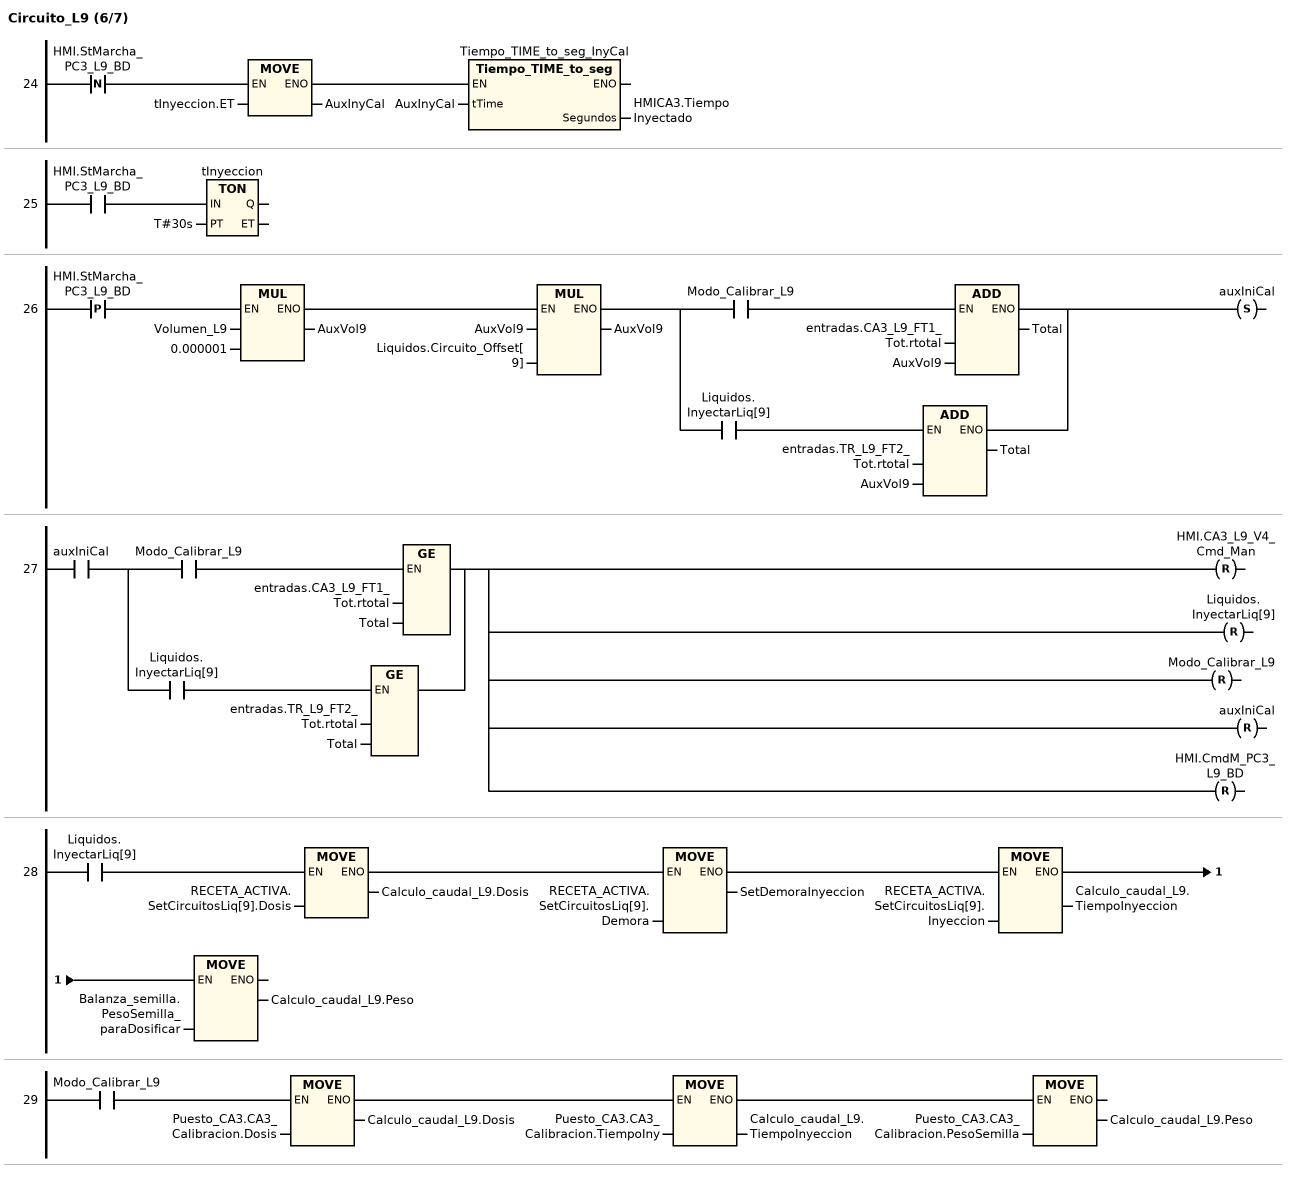
// NETWORK 24
_ft1(CLK := HMI.StMarcha_PC3_L9_BD);
_w8 := _ft1.Q;
IF _w8 THEN AuxInyCal := tInyeccion.ET; END_IF
IF _w8 THEN
    Tiempo_TIME_to_seg_InyCal(tTime := AuxInyCal, Segundos => HMICA3.TiempoInyectado); // Tiempo_TIME_to_seg
END_IF

// NETWORK 25
tInyeccion(IN := HMI.StMarcha_PC3_L9_BD, PT := T#30s); // TON

// NETWORK 26
_rt1(CLK := HMI.StMarcha_PC3_L9_BD);
_w9 := _rt1.Q;
IF _w9 THEN AuxVol9 := Volumen_L9 * 0.000001; END_IF
IF _w9 THEN AuxVol9 := AuxVol9 * Liquidos.Circuito_Offset[9]; END_IF
IF _w9 AND Modo_Calibrar_L9 THEN Total := entradas.CA3_L9_FT1_Tot.rtotal + AuxVol9; END_IF
IF _w9 AND Liquidos.InyectarLiq[9] THEN Total := entradas.TR_L9_FT2_Tot.rtotal + AuxVol9; END_IF
auxIniCal S= _w9 AND Modo_Calibrar_L9 OR _w9 AND Liquidos.InyectarLiq[9];

// NETWORK 27
_w10 := auxIniCal AND Modo_Calibrar_L9 AND entradas.CA3_L9_FT1_Tot.rtotal >= Total OR auxIniCal AND Liquidos.InyectarLiq[9] AND entradas.TR_L9_FT2_Tot.rtotal >= Total;
HMI.CA3_L9_V4_Cmd_Man R= _w10;
Liquidos.InyectarLiq[9] R= _w10;
Modo_Calibrar_L9 R= _w10;
auxIniCal R= _w10;
HMI.CmdM_PC3_L9_BD R= _w10;

// NETWORK 28
_w11 := Liquidos.InyectarLiq[9];
IF _w11 THEN Calculo_caudal_L9.Dosis := RECETA_ACTIVA.SetCircuitosLiq[9].Dosis; END_IF
IF _w11 THEN SetDemoraInyeccion := RECETA_ACTIVA.SetCircuitosLiq[9].Demora; END_IF
IF _w11 THEN Calculo_caudal_L9.TiempoInyeccion := RECETA_ACTIVA.SetCircuitosLiq[9].Inyeccion; END_IF
IF _w11 THEN Calculo_caudal_L9.Peso := Balanza_semilla.PesoSemilla_paraDosificar; END_IF

// NETWORK 29
_w12 := Modo_Calibrar_L9;
IF _w12 THEN Calculo_caudal_L9.Dosis := Puesto_CA3.CA3_Calibracion.Dosis; END_IF
IF _w12 THEN Calculo_caudal_L9.TiempoInyeccion := Puesto_CA3.CA3_Calibracion.TiempoIny; END_IF
IF _w12 THEN Calculo_caudal_L9.Peso := Puesto_CA3.CA3_Calibracion.PesoSemilla; END_IF

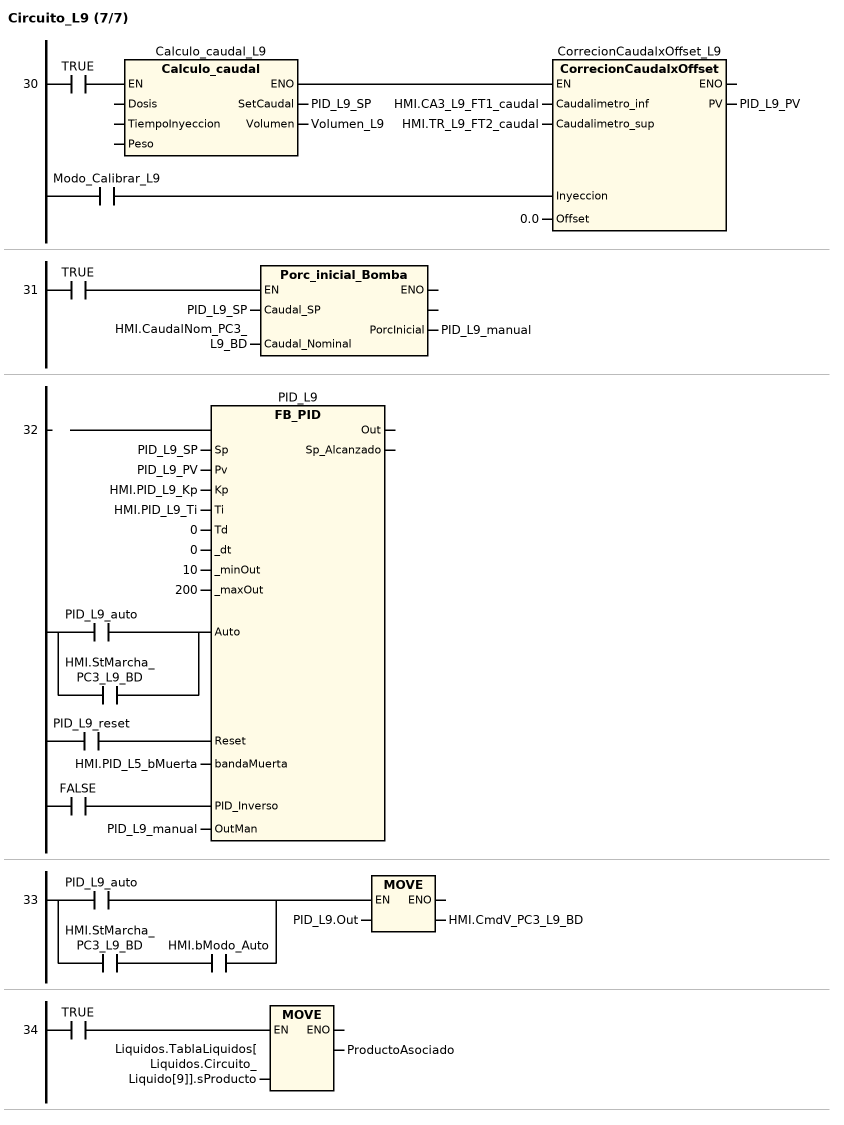
// NETWORK 30
Calculo_caudal_L9(SetCaudal => PID_L9_SP, Volumen => Volumen_L9); // Calculo_caudal
CorrecionCaudalxOffset_L9(
    Caudalimetro_inf := HMI.CA3_L9_FT1_caudal,
    Caudalimetro_sup := HMI.TR_L9_FT2_caudal,
    Inyeccion := Modo_Calibrar_L9,
    Offset := 0.0,
    PV => PID_L9_PV); // CorrecionCaudalxOffset

// NETWORK 31
Porc_inicial_Bomba(Caudal_SP := PID_L9_SP, Caudal_Nominal := HMI.CaudalNom_PC3_L9_BD, PorcInicial => PID_L9_manual);

// NETWORK 32
PID_L9(
    Sp := PID_L9_SP,
    Pv := PID_L9_PV,
    Kp := HMI.PID_L9_Kp,
    Ti := HMI.PID_L9_Ti,
    Td := 0,
    _dt := 0,
    _minOut := 10,
    _maxOut := 200,
    Auto := PID_L9_auto OR HMI.StMarcha_PC3_L9_BD,
    Reset := PID_L9_reset,
    bandaMuerta := HMI.PID_L5_bMuerta,
    PID_Inverso := FALSE,
    OutMan := PID_L9_manual); // FB_PID

// NETWORK 33
IF PID_L9_auto OR HMI.StMarcha_PC3_L9_BD AND HMI.bModo_Auto THEN HMI.CmdV_PC3_L9_BD := PID_L9.Out; END_IF

// NETWORK 34
ProductoAsociado := Liquidos.TablaLiquidos[Liquidos.Circuito_Liquido[9]].sProducto;

END_PROGRAM

// ---- POUs/Puesto_Calibracion_3/Puesto_CA3.TcPOU
PROGRAM Puesto_CA3
VAR
	Balanza_CA3: Balanza;
	dHS:DINT;
	Cmd_Full: R_TRIG;
	TmrLabelFinalizado: TON;
	AuxFinCalibrar:BOOL;
	CA3_Calibracion: Calibracion_Liq_calc;
	Tarar_balanza :BOOL;
	Offset_ref3:REAL;
	Inyectar_ref3:BOOL;
	InicioCal_ref3:BOOL;
	Offset_ref: REAL;
	Inyectar_ref: BOOL;
	InicioCal_ref: BOOL;

	UltimaCalibracao: UDINT;
	VazaoMax: REAL;
	VazaoMaxExcedida: BOOL;
END_VAR

//Indica a ultima calibração da linha selecionada
UltimaCalibracao := HMI.UltimasCalibracoes[HMI.iCircuito_a_calibrar];


Balanza_CA3(
	wStatus:=Entradas.CA3_WT1_wStatus , 
	rValue_REAL:=Entradas.CA3_WT1_rValue_REAL , 
	nValue_DINT:=Entradas.CA3_WT1_nValue_DINT , 
	nValue_Supply:=dHS , 
	nValue_Bridge:=dHS , 
	stEcSlaveAmsNetAdr:=Entradas.CA3_WT1_stEcSlaveAmsNetAdr , 
	bWcState:=Entradas.CA3_WT1_bWcState , 
	wState:=Entradas.CA3_WT1_wState , 
	bCmd_FullCalibration:=HMI.bCmd_Full_WT_CA3 , 
	bCmd_ZeroCalibration:=HMI.bCmd_Zero_WT_CA3 , 
	bCmd_Tara:=Tarar_balanza , 
	bCmd_LoadReference:=HMI.bCmd_LoadReference_WT_CA3 ,
	fLoadReference:=(HMI.rPesoPatron_WT_CA3)/1000,
	wControl=>Salidas.CA3_WT1_wControl );

	TmrLabelFinalizado(IN:= HMI.bCmd_Full_WT_CA3 , PT:=T#10S , Q=> , ET=> );	
	
	HMI.bCmd_LoadReference_WT_CA3:=FALSE;
	HMI.bCmd_Zero_WT_CA3:=FALSE;
	HMI.bCmd_Full_WT_CA3:=FALSE;
	Tarar_balanza:=FALSE;
	Cmd_Full(CLK:=TmrLabelFinalizado.Q , Q=> );
	IF 	Cmd_Full.Q THEN
		HMI.bCalibrado_WT_CA3:=TRUE;
	END_IF	
/////////////////
IF (8<HMI.iCircuito_a_calibrar AND HMI.iCircuito_a_calibrar<13) THEN
//
/////////
CASE HMI.iCircuito_a_calibrar OF
	9:	Offset_ref:=Liquidos.Circuito_Offset[9];
		Inyectar_ref:=circuito_L9.Modo_Calibrar_L9;
		InicioCal_ref:=HMICA3.Inicio_calibracion;
		HMICA3.VolumenPedido_calibracion:=circuito_L9.Volumen_L9;
	10:	Offset_ref:=Liquidos.Circuito_Offset[10];
		Inyectar_ref:=circuito_L10.Modo_Calibrar_L10;
		InicioCal_ref:=HMICA3.Inicio_calibracion;
		HMICA3.VolumenPedido_calibracion:=circuito_L10.Volumen_L10;	
	11:	Offset_ref:=Liquidos.Circuito_Offset[11];
		Inyectar_ref:=circuito_L11.Modo_Calibrar_L11;
		InicioCal_ref:=HMICA3.Inicio_calibracion;
		HMICA3.VolumenPedido_calibracion:=circuito_L11.Volumen_L11;
	12:	Offset_ref:=Liquidos.Circuito_Offset[12];
		Inyectar_ref:=circuito_L12.Modo_Calibrar_L12;
		InicioCal_ref:=HMICA3.Inicio_calibracion;
		HMICA3.VolumenPedido_calibracion:=circuito_L12.Volumen_L12;	
		
		ELSE
	;		
END_CASE
CA3_Calibracion(
	Dosis:=HMICA3.Dosis_calibracion , 
	PesoSemilla:=HMICA3.Peso_calibracion,
	Tolerancia:=HMICA3.Tolerancia_calibracion , 
	PesoBalanza:=Entradas.CA3_WT1_rValue_REAL ,
	mlPedido:= HMICA3.VolumenPedido_calibracion,
	PesoEspec:=Puesto_CA1.PesoEspec , 
	Offset:=Offset_ref ,
	TiempoIny:=HMICA3.TInyeccion_calibracion , 
	Vol_Probeta:=(HMICA3.VolMaxProbeta_calibracion*1000) , 
	Pausa:=HMICA3.Pausa_calibracion , 
	Dosificar=> , 
	Probeta_Llena:=HMICA3.VaciarProbeta_calibracion , 
	Inyectar:=Inyectar_ref, 
	ml:=HMICA3.Volumen_calibracion, 
	Tiempo:=HMICA3.Tiempo_calibracion , 
	InicioCal:= InicioCal_ref, 
	Continuar:=HMICA3.Continuar_calibracion , 
	Tarar:=Tarar_balanza,
	Finalizado:=HMICA3.Fin_calibracion,
	mlProbeta=>HMICA3.Vol_enProbeta , 
	TiempoInyectado:=HMICA3.TiempoInyectado,
	Error_promedio=> HMICA3.Error_promedio, );
//
CASE HMI.iCircuito_a_calibrar OF
	9:	Liquidos.Circuito_Offset[9]:=Offset_ref;//Offset_ref
		circuito_L9.Modo_Calibrar_L9:=Inyectar_ref;//Inyectar_ref
		HMICA3.Inicio_calibracion:=InicioCal_ref;
		VazaoMax := HMI.CaudalNom_PC3_L9_BD;
	10:	Liquidos.Circuito_Offset[10]:=Offset_ref;//Offset_ref
		circuito_L10.Modo_Calibrar_L10:=Inyectar_ref;//Inyectar_ref
		HMICA3.Inicio_calibracion:=InicioCal_ref;
		VazaoMax := HMI.CaudalNom_PC3_L10_BD;
	11:	Liquidos.Circuito_Offset[11]:=Offset_ref;//Offset_ref
		circuito_L11.Modo_Calibrar_L11:=Inyectar_ref;//Inyectar_ref
		HMICA3.Inicio_calibracion:=InicioCal_ref;
		VazaoMax := HMI.CaudalNom_PC3_L11_BD;
	12:	Liquidos.Circuito_Offset[12]:=Offset_ref;//Offset_ref
		circuito_L12.Modo_Calibrar_L12:=Inyectar_ref;//Inyectar_ref
		HMICA3.Inicio_calibracion:=InicioCal_ref;
		VazaoMax := HMI.CaudalNom_PC3_L12_BD;
		
		ELSE
	;		
END_CASE	
END_IF	

IF HMICA3.TInyeccion_calibracion > 0 THEN
	IF (HMICA3.Dosis_calibracion*HMICA3.Peso_calibracion/100)/TO_REAL(HMICA3.TInyeccion_calibracion) > VazaoMax THEN
		VazaoMaxExcedida := TRUE;
	ELSE
		VazaoMaxExcedida := FALSE;
	END_IF
END_IF

END_PROGRAM

// ---- POUs/Puesto_Calibracion_3/Circuito_L10.TcPOU
PROGRAM Circuito_L10
VAR_INPUT
	Modo_Calibrar_L10: BOOL;
END_VAR
VAR
		fbBomba_L10 :Equipo_Motor_ATV320;
		ControlValv_ioLink_V1:ControlValv_ioLink;
		ControlValv_ioLink_V2: ControlValv_ioLink;
		ControlValv_ioLink_V3: ControlValv_ioLink;
		ControlValv_ioLink_V4: ControlValv_ioLink;
		Falla_L10_V1:BOOL;
		Falla_L10_V2:BOOL;
		Falla_L10_V3:BOOL;
		Falla_L10_V4:BOOL;
	Balanza_PU3_WT10: Balanza;
		dHS:DINT;
		TOF_calibradoIBC: TOF;
		PID_L10_SP:REAL;
		PID_L10_auto:BOOL;
		PID_L10_reset:BOOL;
		PID_L10_manual:REAL;
		PID_L10_bMuerta:REAL := 5;
		PID_L10_Kp:REAL := 0.1;
		PID_L10_Ti:REAL := 100;
		PID_L10_PV:REAL;
		Dosis_L10	:REAL;
		TiempoInyeccion_L10	:DINT;
		Peso	:REAL;
		Offset_L10:REAL;
		Inyeccion_L10:BOOL;

		Volumen_L10:REAL;
		Calculo_caudal_L10: Calculo_caudal;
		CorrecionCaudalxOffset_L10: CorrecionCaudalxOffset;
		tInyeccion: TON;
		Total :REAL;
		Totalant	:REAL;
		auxIniCal:BOOL;
		AuxVol10:REAL;
		TDemoraInyectar: TON;
		SetDemoraInyeccion: REAL;
		Tiempo_seg_to_TIME_DemoraInyec: Tiempo_seg_to_TIME;
		AuxTDemoraInyec: TIME;
		PID_L10: FB_PID;
		Tiempo_TIME_to_seg_InyCal: Tiempo_TIME_to_seg;
		AuxInyCal:TIME;
	ProductoAsociado: STRING;
	Lavagem_Circuito10: Lavagem;
END_VAR
VAR PERSISTENT
	UltimaCalibracao	:UDINT;	//Data e hora da ultima calibração
END_VAR
VAR // added by the converter: edge detectors and wires of the graphical bodies
    _w1, _w2, _w3, _w4, _w5, _w6, _w7, _w8, _w9, _w10, _w11, _w12 : BOOL;
    _ft1 : F_TRIG;
    _rt1 : R_TRIG;
END_VAR

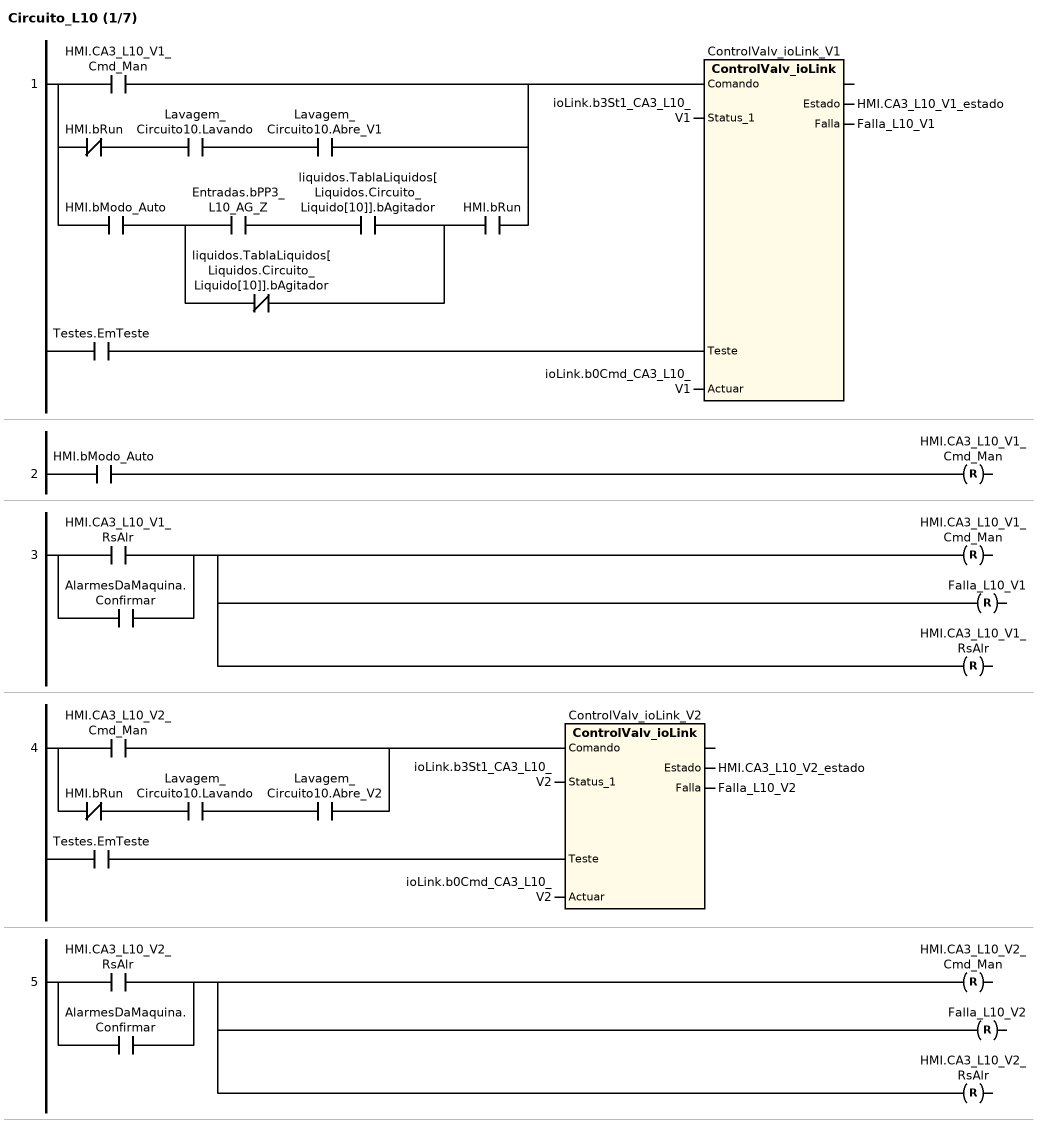
// NETWORK 1
ControlValv_ioLink_V1(
    Comando := HMI.CA3_L10_V1_Cmd_Man OR NOT HMI.bRun AND Lavagem_Circuito10.Lavando AND Lavagem_Circuito10.Abre_V1 OR HMI.bModo_Auto AND (Entradas.bPP3_L10_AG_Z AND (liquidos.TablaLiquidos[Liquidos.Circuito_Liquido[10]].bAgitador) OR NOT (liquidos.TablaLiquidos[Liquidos.Circuito_Liquido[10]].bAgitador)) AND HMI.bRun,
    Status_1 := ioLink.b3St1_CA3_L10_V1,
    Teste := Testes.EmTeste,
    Actuar := ioLink.b0Cmd_CA3_L10_V1,
    Estado => HMI.CA3_L10_V1_estado,
    Falla => Falla_L10_V1); // ControlValv_ioLink

// NETWORK 2
HMI.CA3_L10_V1_Cmd_Man R= HMI.bModo_Auto;

// NETWORK 3
_w1 := HMI.CA3_L10_V1_RsAlr OR AlarmesDaMaquina.Confirmar;
HMI.CA3_L10_V1_Cmd_Man R= _w1;
Falla_L10_V1 R= _w1;
HMI.CA3_L10_V1_RsAlr R= _w1;

// NETWORK 4
ControlValv_ioLink_V2(
    Comando := HMI.CA3_L10_V2_Cmd_Man OR NOT HMI.bRun AND Lavagem_Circuito10.Lavando AND Lavagem_Circuito10.Abre_V2,
    Status_1 := ioLink.b3St1_CA3_L10_V2,
    Teste := Testes.EmTeste,
    Actuar := ioLink.b0Cmd_CA3_L10_V2,
    Estado => HMI.CA3_L10_V2_estado,
    Falla => Falla_L10_V2); // ControlValv_ioLink

// NETWORK 5
_w2 := HMI.CA3_L10_V2_RsAlr OR AlarmesDaMaquina.Confirmar;
HMI.CA3_L10_V2_Cmd_Man R= _w2;
Falla_L10_V2 R= _w2;
HMI.CA3_L10_V2_RsAlr R= _w2;

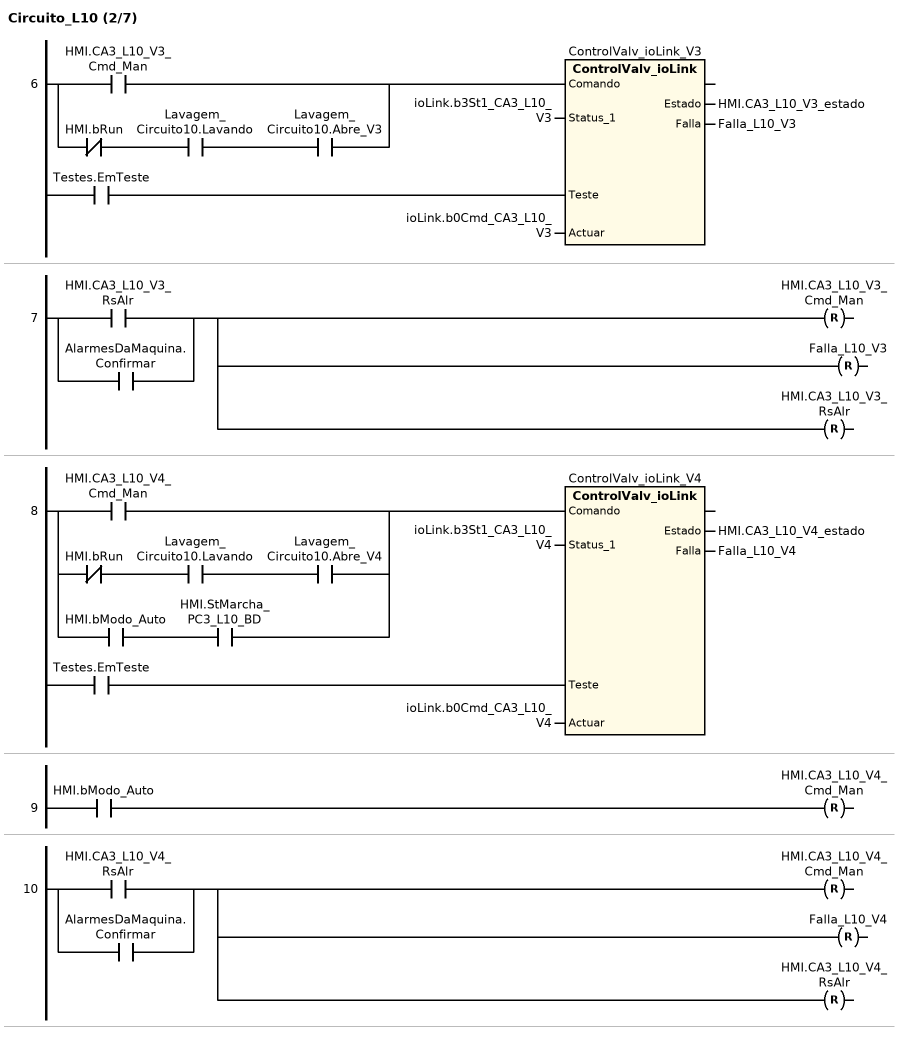
// NETWORK 6
ControlValv_ioLink_V3(
    Comando := HMI.CA3_L10_V3_Cmd_Man OR NOT HMI.bRun AND Lavagem_Circuito10.Lavando AND Lavagem_Circuito10.Abre_V3,
    Status_1 := ioLink.b3St1_CA3_L10_V3,
    Teste := Testes.EmTeste,
    Actuar := ioLink.b0Cmd_CA3_L10_V3,
    Estado => HMI.CA3_L10_V3_estado,
    Falla => Falla_L10_V3); // ControlValv_ioLink

// NETWORK 7
_w3 := HMI.CA3_L10_V3_RsAlr OR AlarmesDaMaquina.Confirmar;
HMI.CA3_L10_V3_Cmd_Man R= _w3;
Falla_L10_V3 R= _w3;
HMI.CA3_L10_V3_RsAlr R= _w3;

// NETWORK 8
ControlValv_ioLink_V4(
    Comando := HMI.CA3_L10_V4_Cmd_Man OR NOT HMI.bRun AND Lavagem_Circuito10.Lavando AND Lavagem_Circuito10.Abre_V4 OR HMI.bModo_Auto AND HMI.StMarcha_PC3_L10_BD,
    Status_1 := ioLink.b3St1_CA3_L10_V4,
    Teste := Testes.EmTeste,
    Actuar := ioLink.b0Cmd_CA3_L10_V4,
    Estado => HMI.CA3_L10_V4_estado,
    Falla => Falla_L10_V4); // ControlValv_ioLink

// NETWORK 9
HMI.CA3_L10_V4_Cmd_Man R= HMI.bModo_Auto;

// NETWORK 10
_w4 := HMI.CA3_L10_V4_RsAlr OR AlarmesDaMaquina.Confirmar;
HMI.CA3_L10_V4_Cmd_Man R= _w4;
Falla_L10_V4 R= _w4;
HMI.CA3_L10_V4_RsAlr R= _w4;

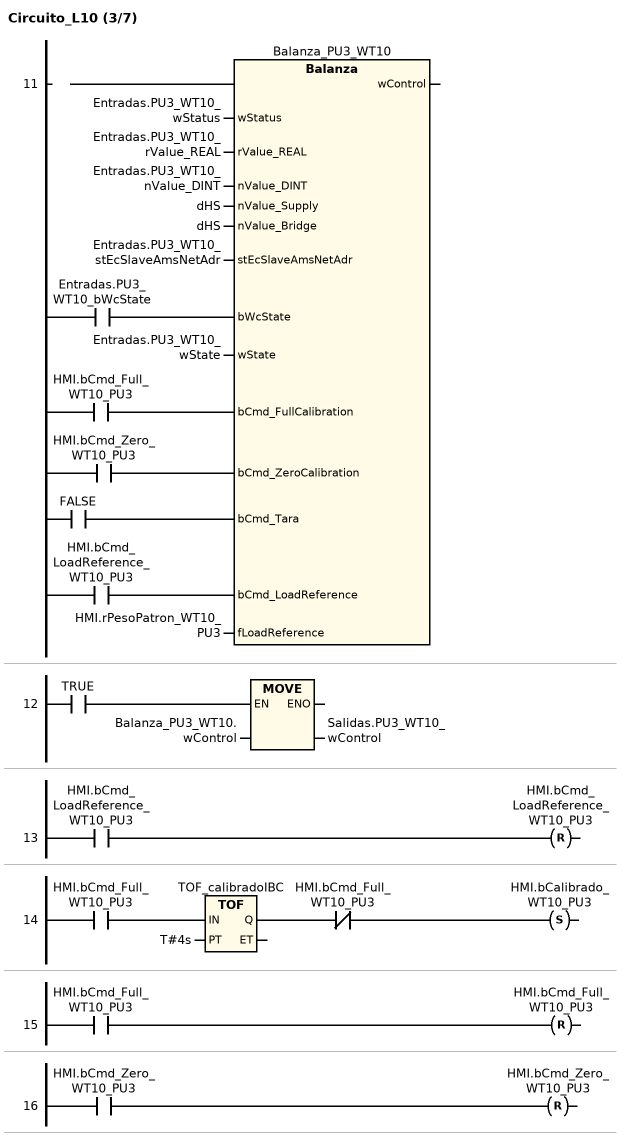
// NETWORK 11
Balanza_PU3_WT10(
    wStatus := Entradas.PU3_WT10_wStatus,
    rValue_REAL := Entradas.PU3_WT10_rValue_REAL,
    nValue_DINT := Entradas.PU3_WT10_nValue_DINT,
    nValue_Supply := dHS,
    nValue_Bridge := dHS,
    stEcSlaveAmsNetAdr := Entradas.PU3_WT10_stEcSlaveAmsNetAdr,
    bWcState := Entradas.PU3_WT10_bWcState,
    wState := Entradas.PU3_WT10_wState,
    bCmd_FullCalibration := HMI.bCmd_Full_WT10_PU3,
    bCmd_ZeroCalibration := HMI.bCmd_Zero_WT10_PU3,
    bCmd_Tara := FALSE,
    bCmd_LoadReference := HMI.bCmd_LoadReference_WT10_PU3,
    fLoadReference := HMI.rPesoPatron_WT10_PU3); // Balanza

// NETWORK 12
Salidas.PU3_WT10_wControl := Balanza_PU3_WT10.wControl;

// NETWORK 13
HMI.bCmd_LoadReference_WT10_PU3 R= HMI.bCmd_LoadReference_WT10_PU3;

// NETWORK 14
TOF_calibradoIBC(IN := HMI.bCmd_Full_WT10_PU3, PT := T#4s); // TOF
HMI.bCalibrado_WT10_PU3 S= TOF_calibradoIBC.Q AND NOT HMI.bCmd_Full_WT10_PU3;

// NETWORK 15
HMI.bCmd_Full_WT10_PU3 R= HMI.bCmd_Full_WT10_PU3;

// NETWORK 16
HMI.bCmd_Zero_WT10_PU3 R= HMI.bCmd_Zero_WT10_PU3;

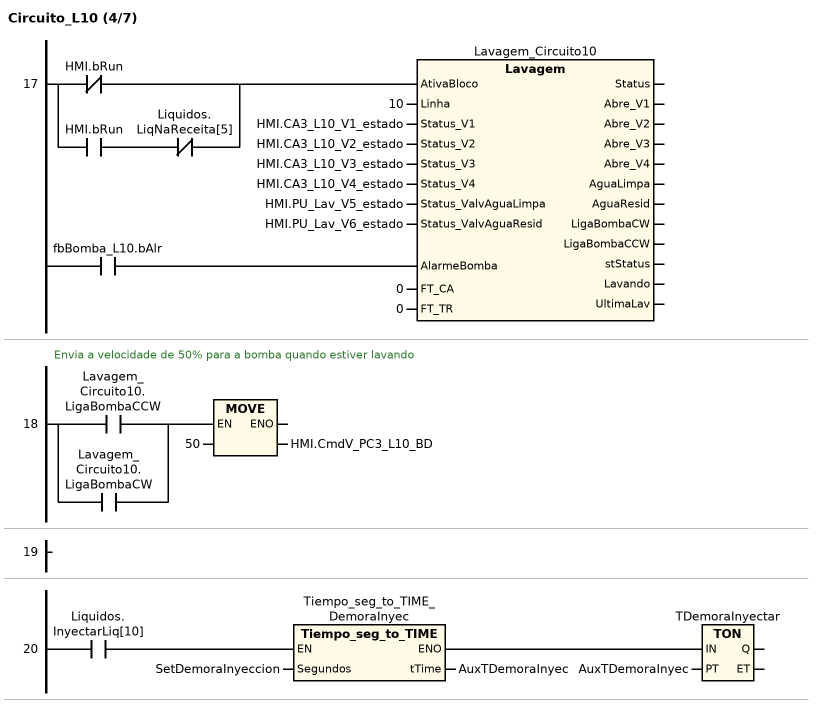
// NETWORK 17
Lavagem_Circuito10(
    AtivaBloco := NOT HMI.bRun OR HMI.bRun AND NOT Liquidos.LiqNaReceita[5],
    Linha := 10,
    Status_V1 := HMI.CA3_L10_V1_estado,
    Status_V2 := HMI.CA3_L10_V2_estado,
    Status_V3 := HMI.CA3_L10_V3_estado,
    Status_V4 := HMI.CA3_L10_V4_estado,
    Status_ValvAguaLimpa := HMI.PU_Lav_V5_estado,
    Status_ValvAguaResid := HMI.PU_Lav_V6_estado,
    AlarmeBomba := fbBomba_L10.bAlr,
    FT_CA := 0,
    FT_TR := 0); // Lavagem

// NETWORK 18
// Envia a velocidade de 50% para a bomba quando estiver lavando
IF Lavagem_Circuito10.LigaBombaCCW OR Lavagem_Circuito10.LigaBombaCW THEN HMI.CmdV_PC3_L10_BD := 50; END_IF

// NETWORK 19

// NETWORK 20
_w5 := Liquidos.InyectarLiq[10];
IF _w5 THEN
    Tiempo_seg_to_TIME_DemoraInyec(Segundos := SetDemoraInyeccion, tTime => AuxTDemoraInyec); // Tiempo_seg_to_TIME
END_IF
TDemoraInyectar(IN := _w5, PT := AuxTDemoraInyec); // TON

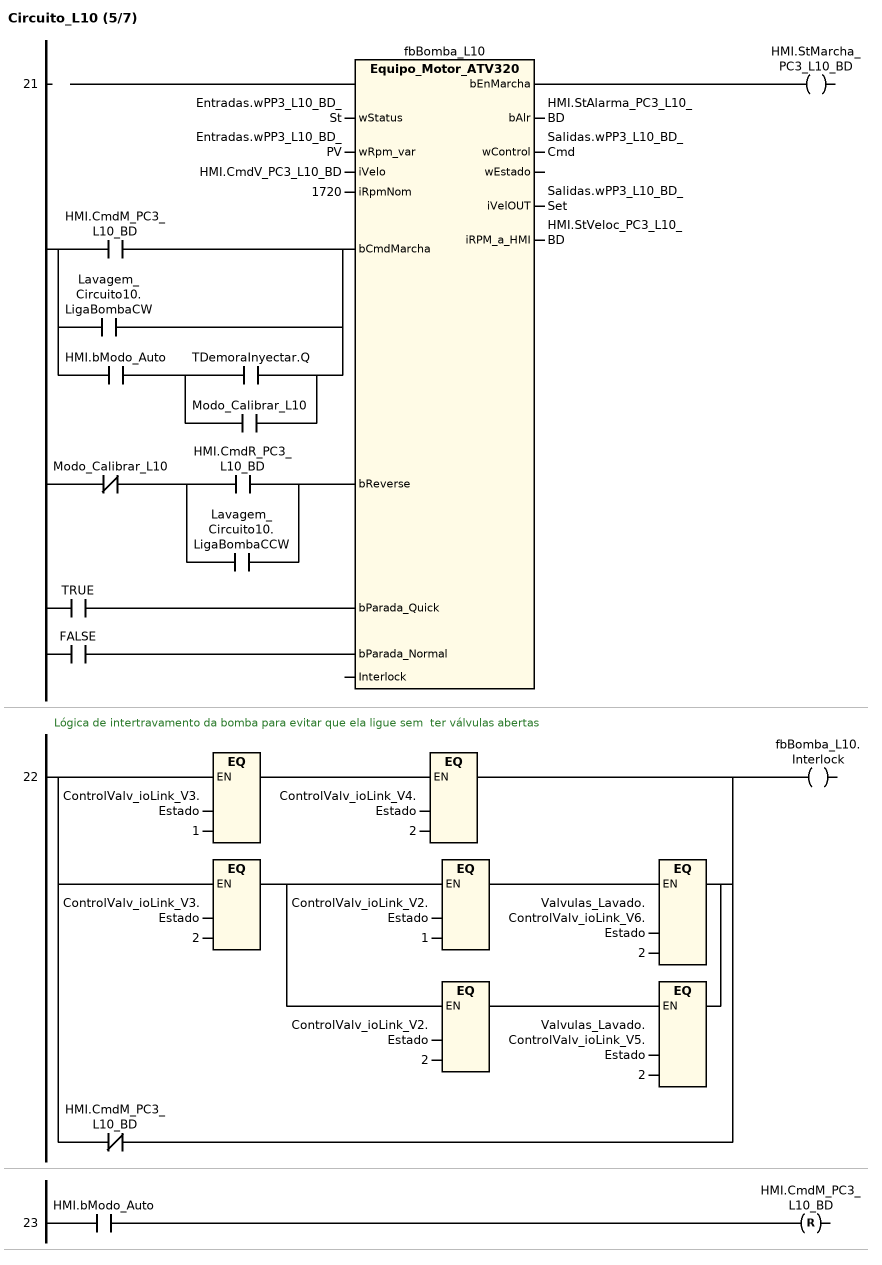
// NETWORK 21
fbBomba_L10(
    wStatus := Entradas.wPP3_L10_BD_St,
    wRpm_var := Entradas.wPP3_L10_BD_PV,
    iVelo := HMI.CmdV_PC3_L10_BD,
    iRpmNom := 1720,
    bCmdMarcha := HMI.CmdM_PC3_L10_BD OR Lavagem_Circuito10.LigaBombaCW OR HMI.bModo_Auto AND (TDemoraInyectar.Q OR Modo_Calibrar_L10),
    bReverse := NOT Modo_Calibrar_L10 AND (HMI.CmdR_PC3_L10_BD OR Lavagem_Circuito10.LigaBombaCCW),
    bParada_Quick := TRUE,
    bParada_Normal := FALSE,
    bAlr => HMI.StAlarma_PC3_L10_BD,
    wControl => Salidas.wPP3_L10_BD_Cmd,
    iVelOUT => Salidas.wPP3_L10_BD_Set,
    iRPM_a_HMI => HMI.StVeloc_PC3_L10_BD); // Equipo_Motor_ATV320
HMI.StMarcha_PC3_L10_BD := fbBomba_L10.bEnMarcha;

// NETWORK 22
// Lógica de intertravamento da bomba para evitar que ela ligue sem  ter válvulas abertas
_w6 := NOT HMI.CmdM_PC3_L10_BD;
IF NOT _w6 THEN
    _w7 := ControlValv_ioLink_V3.Estado = 2;
    _w6 := ControlValv_ioLink_V3.Estado = 1 AND ControlValv_ioLink_V4.Estado = 2 OR (_w7 AND ControlValv_ioLink_V2.Estado = 1 AND Valvulas_Lavado.ControlValv_ioLink_V6.Estado = 2 OR _w7 AND ControlValv_ioLink_V2.Estado = 2 AND Valvulas_Lavado.ControlValv_ioLink_V5.Estado = 2);
END_IF
fbBomba_L10.Interlock := _w6;

// NETWORK 23
HMI.CmdM_PC3_L10_BD R= HMI.bModo_Auto;

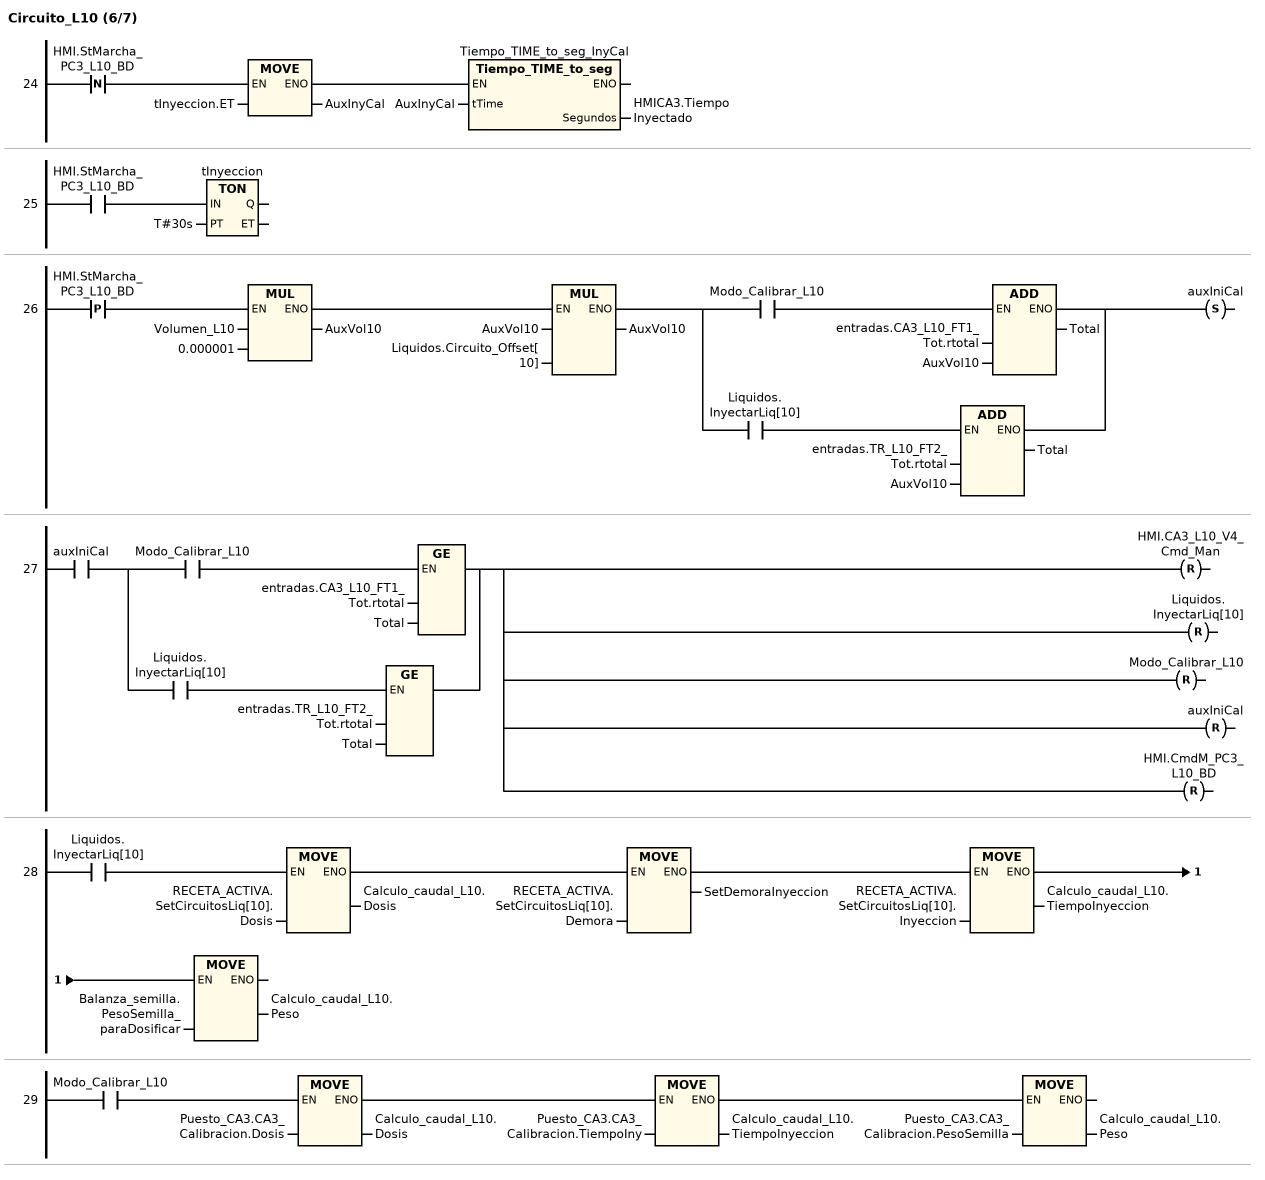
// NETWORK 24
_ft1(CLK := HMI.StMarcha_PC3_L10_BD);
_w8 := _ft1.Q;
IF _w8 THEN AuxInyCal := tInyeccion.ET; END_IF
IF _w8 THEN
    Tiempo_TIME_to_seg_InyCal(tTime := AuxInyCal, Segundos => HMICA3.TiempoInyectado); // Tiempo_TIME_to_seg
END_IF

// NETWORK 25
tInyeccion(IN := HMI.StMarcha_PC3_L10_BD, PT := T#30s); // TON

// NETWORK 26
_rt1(CLK := HMI.StMarcha_PC3_L10_BD);
_w9 := _rt1.Q;
IF _w9 THEN AuxVol10 := Volumen_L10 * 0.000001; END_IF
IF _w9 THEN AuxVol10 := AuxVol10 * Liquidos.Circuito_Offset[10]; END_IF
IF _w9 AND Modo_Calibrar_L10 THEN Total := entradas.CA3_L10_FT1_Tot.rtotal + AuxVol10; END_IF
IF _w9 AND Liquidos.InyectarLiq[10] THEN Total := entradas.TR_L10_FT2_Tot.rtotal + AuxVol10; END_IF
auxIniCal S= _w9 AND Modo_Calibrar_L10 OR _w9 AND Liquidos.InyectarLiq[10];

// NETWORK 27
_w10 := auxIniCal AND Modo_Calibrar_L10 AND entradas.CA3_L10_FT1_Tot.rtotal >= Total OR auxIniCal AND Liquidos.InyectarLiq[10] AND entradas.TR_L10_FT2_Tot.rtotal >= Total;
HMI.CA3_L10_V4_Cmd_Man R= _w10;
Liquidos.InyectarLiq[10] R= _w10;
Modo_Calibrar_L10 R= _w10;
auxIniCal R= _w10;
HMI.CmdM_PC3_L10_BD R= _w10;

// NETWORK 28
_w11 := Liquidos.InyectarLiq[10];
IF _w11 THEN Calculo_caudal_L10.Dosis := RECETA_ACTIVA.SetCircuitosLiq[10].Dosis; END_IF
IF _w11 THEN SetDemoraInyeccion := RECETA_ACTIVA.SetCircuitosLiq[10].Demora; END_IF
IF _w11 THEN Calculo_caudal_L10.TiempoInyeccion := RECETA_ACTIVA.SetCircuitosLiq[10].Inyeccion; END_IF
IF _w11 THEN Calculo_caudal_L10.Peso := Balanza_semilla.PesoSemilla_paraDosificar; END_IF

// NETWORK 29
_w12 := Modo_Calibrar_L10;
IF _w12 THEN Calculo_caudal_L10.Dosis := Puesto_CA3.CA3_Calibracion.Dosis; END_IF
IF _w12 THEN Calculo_caudal_L10.TiempoInyeccion := Puesto_CA3.CA3_Calibracion.TiempoIny; END_IF
IF _w12 THEN Calculo_caudal_L10.Peso := Puesto_CA3.CA3_Calibracion.PesoSemilla; END_IF

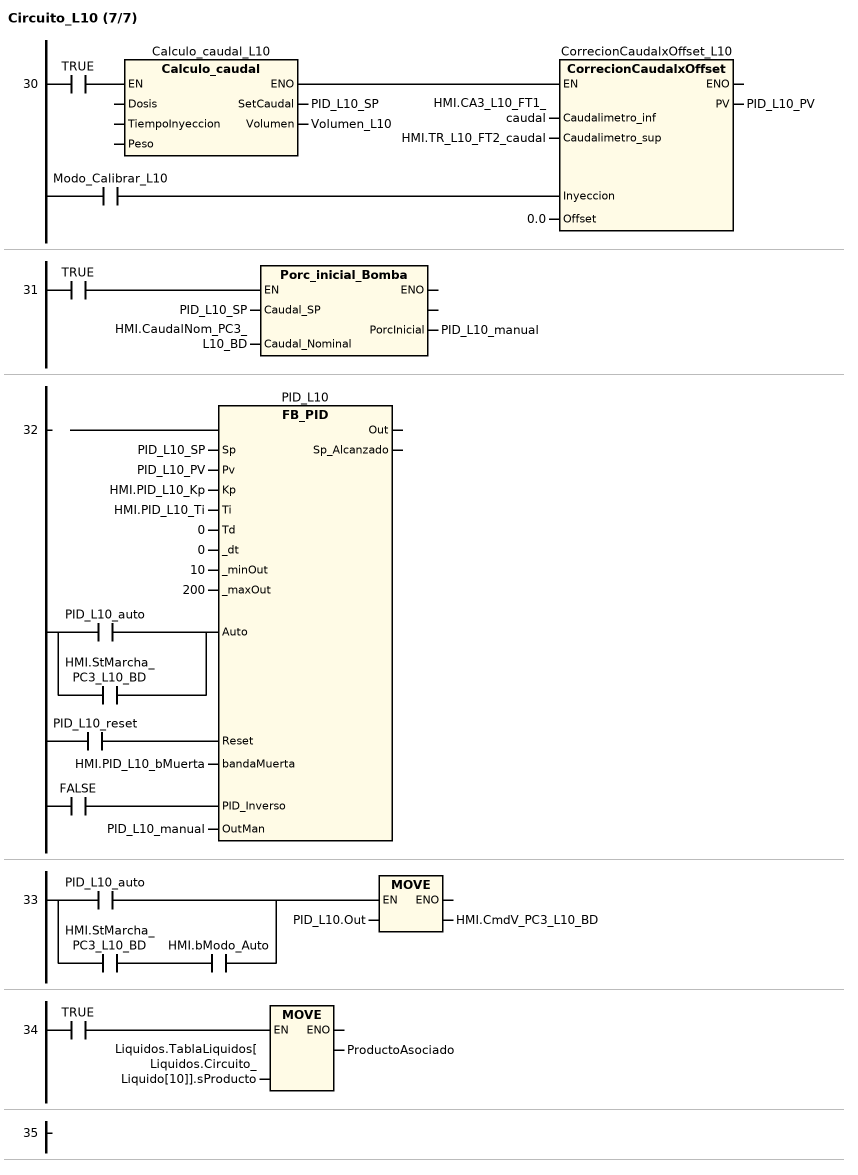
// NETWORK 30
Calculo_caudal_L10(SetCaudal => PID_L10_SP, Volumen => Volumen_L10); // Calculo_caudal
CorrecionCaudalxOffset_L10(
    Caudalimetro_inf := HMI.CA3_L10_FT1_caudal,
    Caudalimetro_sup := HMI.TR_L10_FT2_caudal,
    Inyeccion := Modo_Calibrar_L10,
    Offset := 0.0,
    PV => PID_L10_PV); // CorrecionCaudalxOffset

// NETWORK 31
Porc_inicial_Bomba(Caudal_SP := PID_L10_SP, Caudal_Nominal := HMI.CaudalNom_PC3_L10_BD, PorcInicial => PID_L10_manual);

// NETWORK 32
PID_L10(
    Sp := PID_L10_SP,
    Pv := PID_L10_PV,
    Kp := HMI.PID_L10_Kp,
    Ti := HMI.PID_L10_Ti,
    Td := 0,
    _dt := 0,
    _minOut := 10,
    _maxOut := 200,
    Auto := PID_L10_auto OR HMI.StMarcha_PC3_L10_BD,
    Reset := PID_L10_reset,
    bandaMuerta := HMI.PID_L10_bMuerta,
    PID_Inverso := FALSE,
    OutMan := PID_L10_manual); // FB_PID

// NETWORK 33
IF PID_L10_auto OR HMI.StMarcha_PC3_L10_BD AND HMI.bModo_Auto THEN HMI.CmdV_PC3_L10_BD := PID_L10.Out; END_IF

// NETWORK 34
ProductoAsociado := Liquidos.TablaLiquidos[Liquidos.Circuito_Liquido[10]].sProducto;

// NETWORK 35

END_PROGRAM

// ---- POUs/Puesto_Calibracion_3/Circuito_L11.TcPOU
PROGRAM Circuito_L11
VAR_INPUT
	Modo_Calibrar_L11: BOOL;
END_VAR
VAR
		fbBomba_L11 :Equipo_Motor_ATV320;
		ControlValv_ioLink_V1:ControlValv_ioLink;
		ControlValv_ioLink_V2: ControlValv_ioLink;
		ControlValv_ioLink_V3: ControlValv_ioLink;
		ControlValv_ioLink_V4: ControlValv_ioLink;
		Falla_L11_V1:BOOL;
		Falla_L11_V2:BOOL;
		Falla_L11_V3:BOOL;
		Falla_L11_V4:BOOL;
	Balanza_PU3_WT11: Balanza;
		dHS:DINT;
		TOF_calibradoIBC: TOF;
		PID_L11_SP:REAL;
		PID_L11_auto:BOOL;
		PID_L11_reset:BOOL;
		PID_L11_manual:REAL;
		PID_L11_bMuerta:REAL := 5;
		PID_L11_Kp:REAL := 0.1;
		PID_L11_Ti:REAL := 100;
		PID_L11_PV:REAL;
		Dosis_L11	:REAL;
		TiempoInyeccion_L11	:DINT;
		Peso	:REAL;
		Offset_L11:REAL;
		Inyeccion_L11:BOOL;

		Volumen_L11:REAL;
		Calculo_caudal_L11: Calculo_caudal;
		CorrecionCaudalxOffset_L11: CorrecionCaudalxOffset;
		tInyeccion: TON;
		Total :REAL;
		Totalant	:REAL;
		auxIniCal:BOOL;
		AuxVol11:REAL;
		TDemoraInyectar: TON;
		SetDemoraInyeccion: REAL;
		Tiempo_seg_to_TIME_DemoraInyec: Tiempo_seg_to_TIME;
		AuxTDemoraInyec: TIME;
		PID_L11: FB_PID;
		Tiempo_TIME_to_seg_InyCal: Tiempo_TIME_to_seg;
		AuxInyCal:TIME;		
		IniTotalFT2:REAL;
		Auxconsumo:REAL;
	ProductoAsociado: STRING;
	Lavagem_Circuito11: Lavagem;
END_VAR
VAR PERSISTENT
	UltimaCalibracao	:UDINT;	//Data e hora da ultima calibração
END_VAR
VAR // added by the converter: edge detectors and wires of the graphical bodies
    _w1, _w2, _w3, _w4, _w5, _w6, _w7, _w8, _w9, _w10, _w11, _w12, _w13 : BOOL;
    _ft1 : F_TRIG;
    _rt1, _rt2 : R_TRIG;
END_VAR

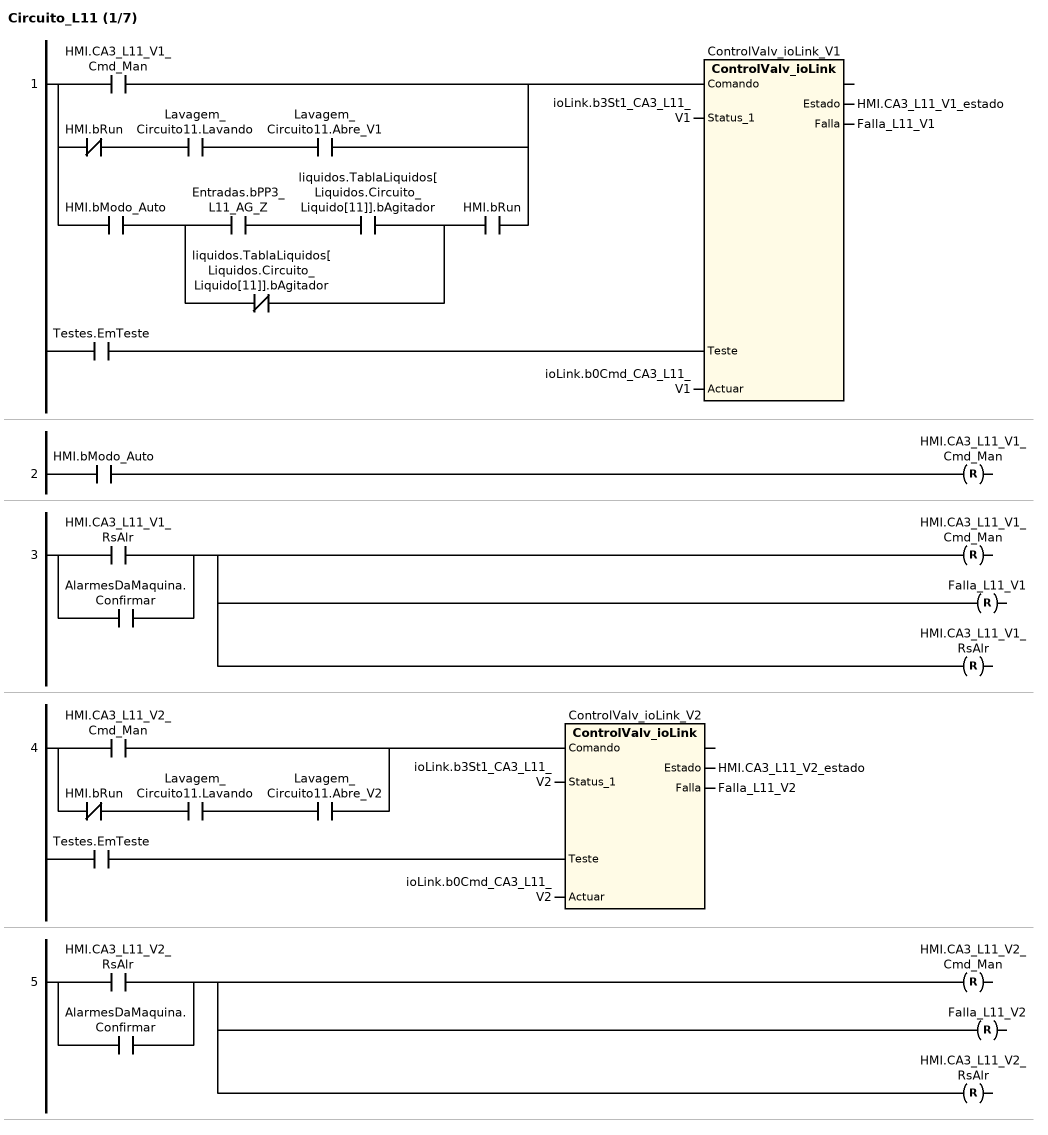
// NETWORK 1
ControlValv_ioLink_V1(
    Comando := HMI.CA3_L11_V1_Cmd_Man OR NOT HMI.bRun AND Lavagem_Circuito11.Lavando AND Lavagem_Circuito11.Abre_V1 OR HMI.bModo_Auto AND (Entradas.bPP3_L11_AG_Z AND (liquidos.TablaLiquidos[Liquidos.Circuito_Liquido[11]].bAgitador) OR NOT (liquidos.TablaLiquidos[Liquidos.Circuito_Liquido[11]].bAgitador)) AND HMI.bRun,
    Status_1 := ioLink.b3St1_CA3_L11_V1,
    Teste := Testes.EmTeste,
    Actuar := ioLink.b0Cmd_CA3_L11_V1,
    Estado => HMI.CA3_L11_V1_estado,
    Falla => Falla_L11_V1); // ControlValv_ioLink

// NETWORK 2
HMI.CA3_L11_V1_Cmd_Man R= HMI.bModo_Auto;

// NETWORK 3
_w1 := HMI.CA3_L11_V1_RsAlr OR AlarmesDaMaquina.Confirmar;
HMI.CA3_L11_V1_Cmd_Man R= _w1;
Falla_L11_V1 R= _w1;
HMI.CA3_L11_V1_RsAlr R= _w1;

// NETWORK 4
ControlValv_ioLink_V2(
    Comando := HMI.CA3_L11_V2_Cmd_Man OR NOT HMI.bRun AND Lavagem_Circuito11.Lavando AND Lavagem_Circuito11.Abre_V2,
    Status_1 := ioLink.b3St1_CA3_L11_V2,
    Teste := Testes.EmTeste,
    Actuar := ioLink.b0Cmd_CA3_L11_V2,
    Estado => HMI.CA3_L11_V2_estado,
    Falla => Falla_L11_V2); // ControlValv_ioLink

// NETWORK 5
_w2 := HMI.CA3_L11_V2_RsAlr OR AlarmesDaMaquina.Confirmar;
HMI.CA3_L11_V2_Cmd_Man R= _w2;
Falla_L11_V2 R= _w2;
HMI.CA3_L11_V2_RsAlr R= _w2;

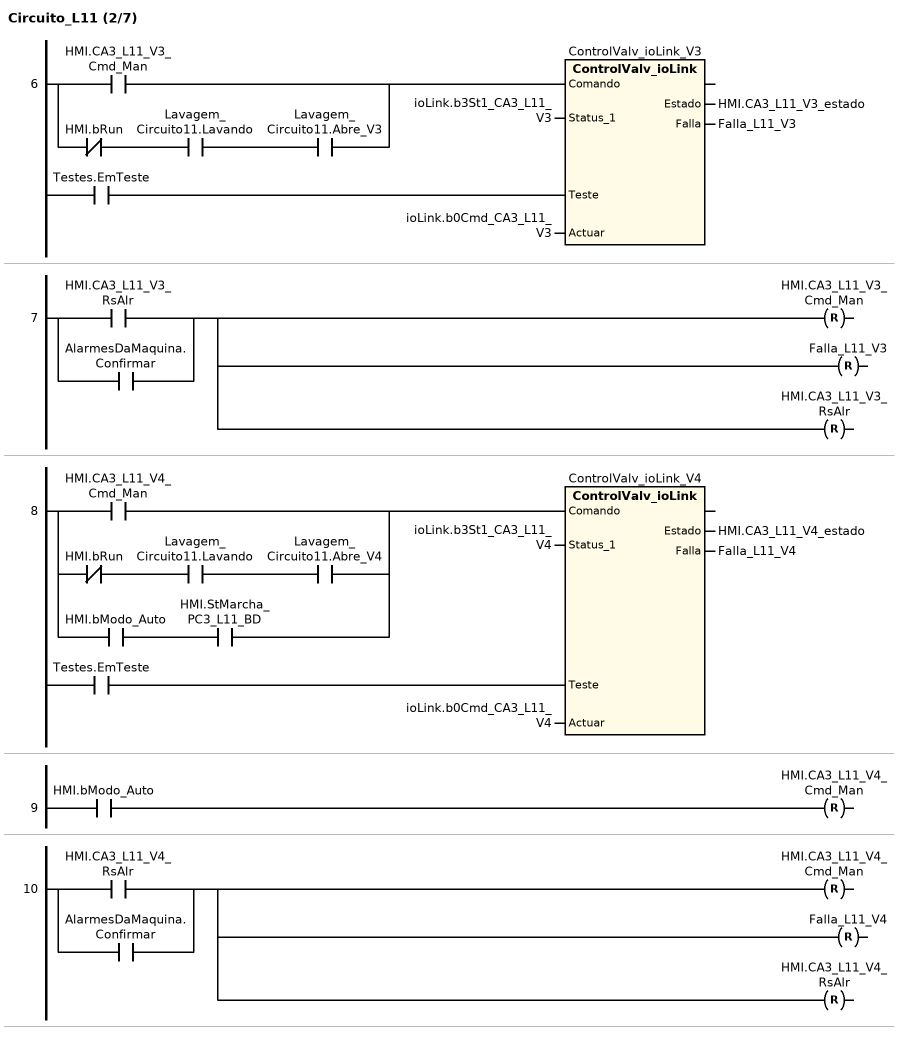
// NETWORK 6
ControlValv_ioLink_V3(
    Comando := HMI.CA3_L11_V3_Cmd_Man OR NOT HMI.bRun AND Lavagem_Circuito11.Lavando AND Lavagem_Circuito11.Abre_V3,
    Status_1 := ioLink.b3St1_CA3_L11_V3,
    Teste := Testes.EmTeste,
    Actuar := ioLink.b0Cmd_CA3_L11_V3,
    Estado => HMI.CA3_L11_V3_estado,
    Falla => Falla_L11_V3); // ControlValv_ioLink

// NETWORK 7
_w3 := HMI.CA3_L11_V3_RsAlr OR AlarmesDaMaquina.Confirmar;
HMI.CA3_L11_V3_Cmd_Man R= _w3;
Falla_L11_V3 R= _w3;
HMI.CA3_L11_V3_RsAlr R= _w3;

// NETWORK 8
ControlValv_ioLink_V4(
    Comando := HMI.CA3_L11_V4_Cmd_Man OR NOT HMI.bRun AND Lavagem_Circuito11.Lavando AND Lavagem_Circuito11.Abre_V4 OR HMI.bModo_Auto AND HMI.StMarcha_PC3_L11_BD,
    Status_1 := ioLink.b3St1_CA3_L11_V4,
    Teste := Testes.EmTeste,
    Actuar := ioLink.b0Cmd_CA3_L11_V4,
    Estado => HMI.CA3_L11_V4_estado,
    Falla => Falla_L11_V4); // ControlValv_ioLink

// NETWORK 9
HMI.CA3_L11_V4_Cmd_Man R= HMI.bModo_Auto;

// NETWORK 10
_w4 := HMI.CA3_L11_V4_RsAlr OR AlarmesDaMaquina.Confirmar;
HMI.CA3_L11_V4_Cmd_Man R= _w4;
Falla_L11_V4 R= _w4;
HMI.CA3_L11_V4_RsAlr R= _w4;

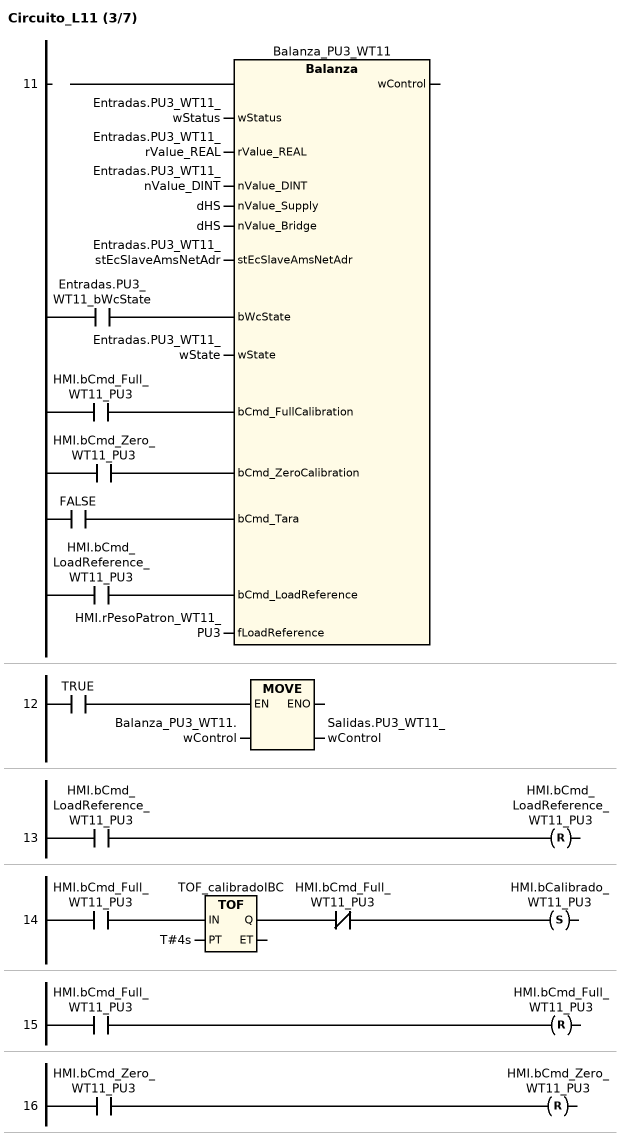
// NETWORK 11
Balanza_PU3_WT11(
    wStatus := Entradas.PU3_WT11_wStatus,
    rValue_REAL := Entradas.PU3_WT11_rValue_REAL,
    nValue_DINT := Entradas.PU3_WT11_nValue_DINT,
    nValue_Supply := dHS,
    nValue_Bridge := dHS,
    stEcSlaveAmsNetAdr := Entradas.PU3_WT11_stEcSlaveAmsNetAdr,
    bWcState := Entradas.PU3_WT11_bWcState,
    wState := Entradas.PU3_WT11_wState,
    bCmd_FullCalibration := HMI.bCmd_Full_WT11_PU3,
    bCmd_ZeroCalibration := HMI.bCmd_Zero_WT11_PU3,
    bCmd_Tara := FALSE,
    bCmd_LoadReference := HMI.bCmd_LoadReference_WT11_PU3,
    fLoadReference := HMI.rPesoPatron_WT11_PU3); // Balanza

// NETWORK 12
Salidas.PU3_WT11_wControl := Balanza_PU3_WT11.wControl;

// NETWORK 13
HMI.bCmd_LoadReference_WT11_PU3 R= HMI.bCmd_LoadReference_WT11_PU3;

// NETWORK 14
TOF_calibradoIBC(IN := HMI.bCmd_Full_WT11_PU3, PT := T#4s); // TOF
HMI.bCalibrado_WT11_PU3 S= TOF_calibradoIBC.Q AND NOT HMI.bCmd_Full_WT11_PU3;

// NETWORK 15
HMI.bCmd_Full_WT11_PU3 R= HMI.bCmd_Full_WT11_PU3;

// NETWORK 16
HMI.bCmd_Zero_WT11_PU3 R= HMI.bCmd_Zero_WT11_PU3;

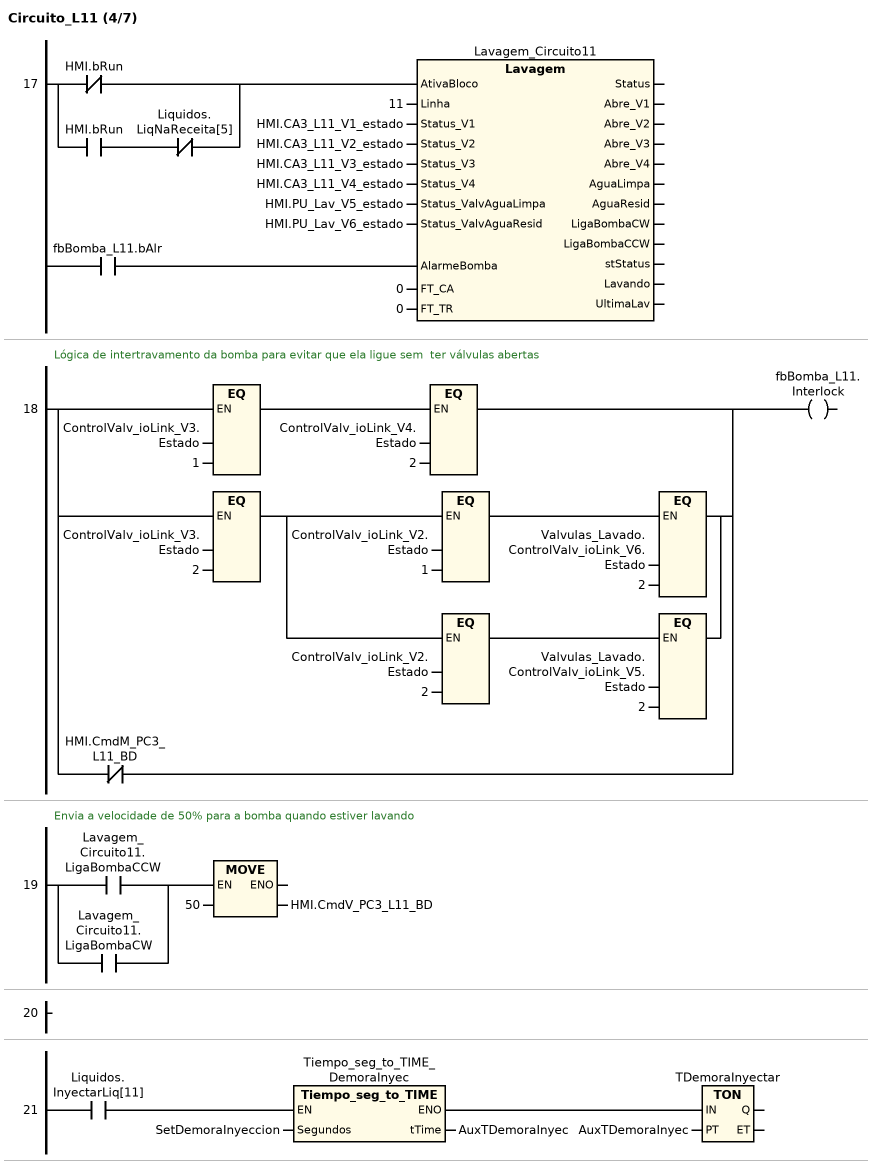
// NETWORK 17
Lavagem_Circuito11(
    AtivaBloco := NOT HMI.bRun OR HMI.bRun AND NOT Liquidos.LiqNaReceita[5],
    Linha := 11,
    Status_V1 := HMI.CA3_L11_V1_estado,
    Status_V2 := HMI.CA3_L11_V2_estado,
    Status_V3 := HMI.CA3_L11_V3_estado,
    Status_V4 := HMI.CA3_L11_V4_estado,
    Status_ValvAguaLimpa := HMI.PU_Lav_V5_estado,
    Status_ValvAguaResid := HMI.PU_Lav_V6_estado,
    AlarmeBomba := fbBomba_L11.bAlr,
    FT_CA := 0,
    FT_TR := 0); // Lavagem

// NETWORK 18
// Lógica de intertravamento da bomba para evitar que ela ligue sem  ter válvulas abertas
_w5 := NOT HMI.CmdM_PC3_L11_BD;
IF NOT _w5 THEN
    _w6 := ControlValv_ioLink_V3.Estado = 2;
    _w5 := ControlValv_ioLink_V3.Estado = 1 AND ControlValv_ioLink_V4.Estado = 2 OR (_w6 AND ControlValv_ioLink_V2.Estado = 1 AND Valvulas_Lavado.ControlValv_ioLink_V6.Estado = 2 OR _w6 AND ControlValv_ioLink_V2.Estado = 2 AND Valvulas_Lavado.ControlValv_ioLink_V5.Estado = 2);
END_IF
fbBomba_L11.Interlock := _w5;

// NETWORK 19
// Envia a velocidade de 50% para a bomba quando estiver lavando
IF Lavagem_Circuito11.LigaBombaCCW OR Lavagem_Circuito11.LigaBombaCW THEN HMI.CmdV_PC3_L11_BD := 50; END_IF

// NETWORK 20

// NETWORK 21
_w7 := Liquidos.InyectarLiq[11];
IF _w7 THEN
    Tiempo_seg_to_TIME_DemoraInyec(Segundos := SetDemoraInyeccion, tTime => AuxTDemoraInyec); // Tiempo_seg_to_TIME
END_IF
TDemoraInyectar(IN := _w7, PT := AuxTDemoraInyec); // TON

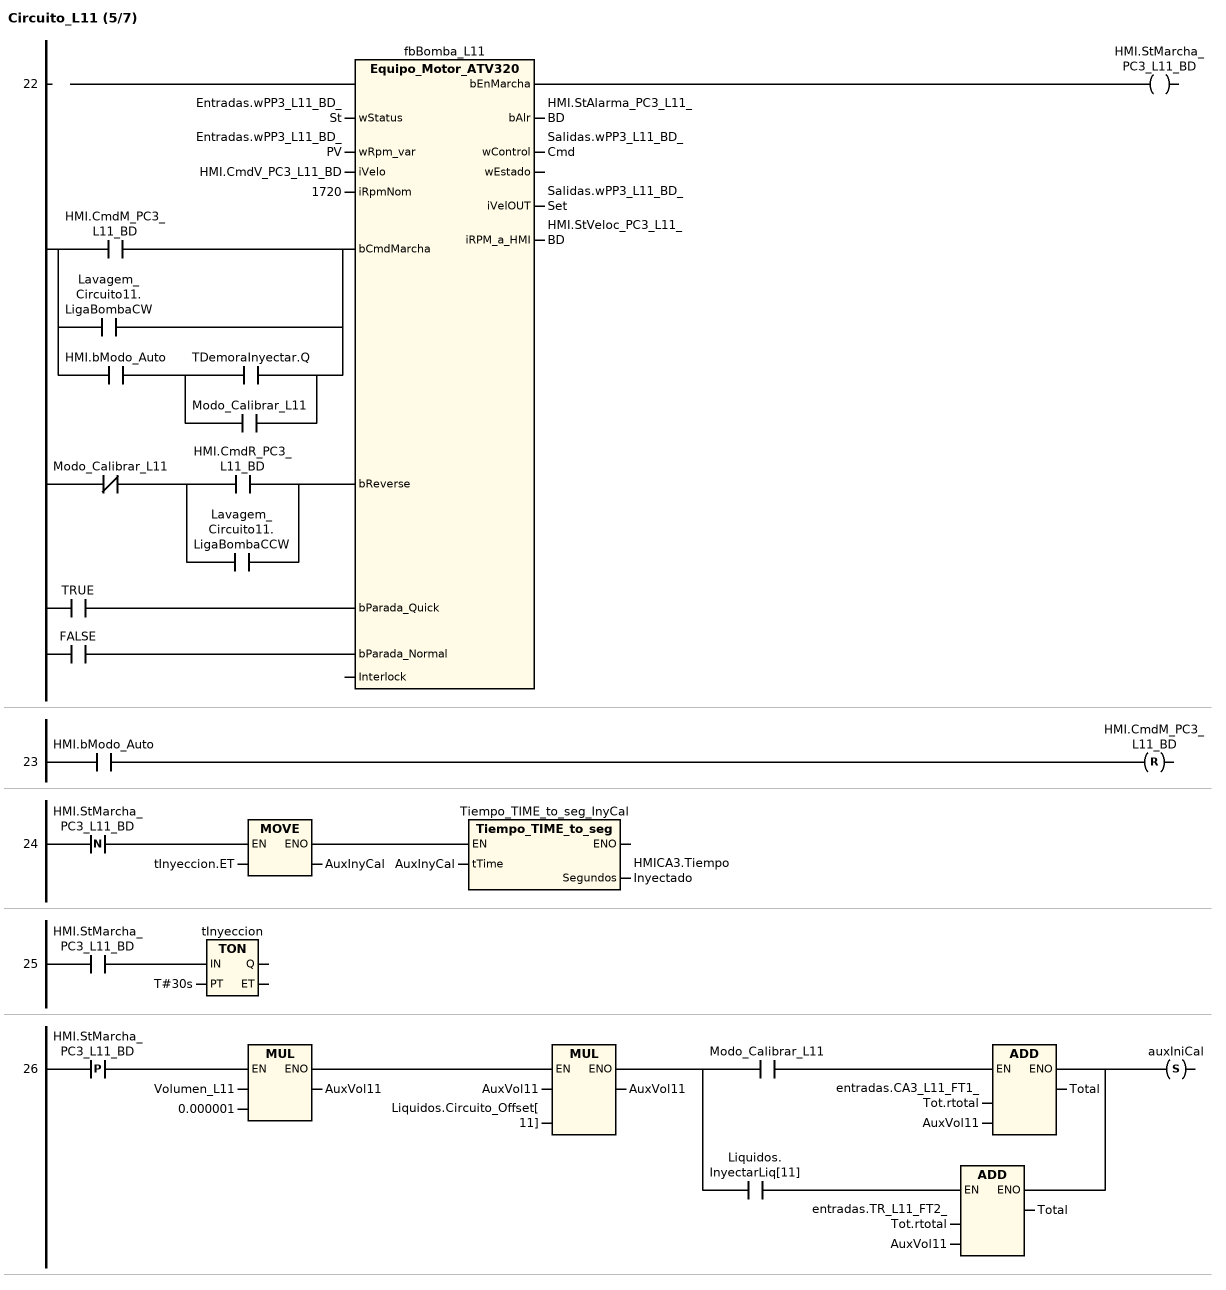
// NETWORK 22
fbBomba_L11(
    wStatus := Entradas.wPP3_L11_BD_St,
    wRpm_var := Entradas.wPP3_L11_BD_PV,
    iVelo := HMI.CmdV_PC3_L11_BD,
    iRpmNom := 1720,
    bCmdMarcha := HMI.CmdM_PC3_L11_BD OR Lavagem_Circuito11.LigaBombaCW OR HMI.bModo_Auto AND (TDemoraInyectar.Q OR Modo_Calibrar_L11),
    bReverse := NOT Modo_Calibrar_L11 AND (HMI.CmdR_PC3_L11_BD OR Lavagem_Circuito11.LigaBombaCCW),
    bParada_Quick := TRUE,
    bParada_Normal := FALSE,
    bAlr => HMI.StAlarma_PC3_L11_BD,
    wControl => Salidas.wPP3_L11_BD_Cmd,
    iVelOUT => Salidas.wPP3_L11_BD_Set,
    iRPM_a_HMI => HMI.StVeloc_PC3_L11_BD); // Equipo_Motor_ATV320
HMI.StMarcha_PC3_L11_BD := fbBomba_L11.bEnMarcha;

// NETWORK 23
HMI.CmdM_PC3_L11_BD R= HMI.bModo_Auto;

// NETWORK 24
_ft1(CLK := HMI.StMarcha_PC3_L11_BD);
_w8 := _ft1.Q;
IF _w8 THEN AuxInyCal := tInyeccion.ET; END_IF
IF _w8 THEN
    Tiempo_TIME_to_seg_InyCal(tTime := AuxInyCal, Segundos => HMICA3.TiempoInyectado); // Tiempo_TIME_to_seg
END_IF

// NETWORK 25
tInyeccion(IN := HMI.StMarcha_PC3_L11_BD, PT := T#30s); // TON

// NETWORK 26
_rt1(CLK := HMI.StMarcha_PC3_L11_BD);
_w9 := _rt1.Q;
IF _w9 THEN AuxVol11 := Volumen_L11 * 0.000001; END_IF
IF _w9 THEN AuxVol11 := AuxVol11 * Liquidos.Circuito_Offset[11]; END_IF
IF _w9 AND Modo_Calibrar_L11 THEN Total := entradas.CA3_L11_FT1_Tot.rtotal + AuxVol11; END_IF
IF _w9 AND Liquidos.InyectarLiq[11] THEN Total := entradas.TR_L11_FT2_Tot.rtotal + AuxVol11; END_IF
auxIniCal S= _w9 AND Modo_Calibrar_L11 OR _w9 AND Liquidos.InyectarLiq[11];

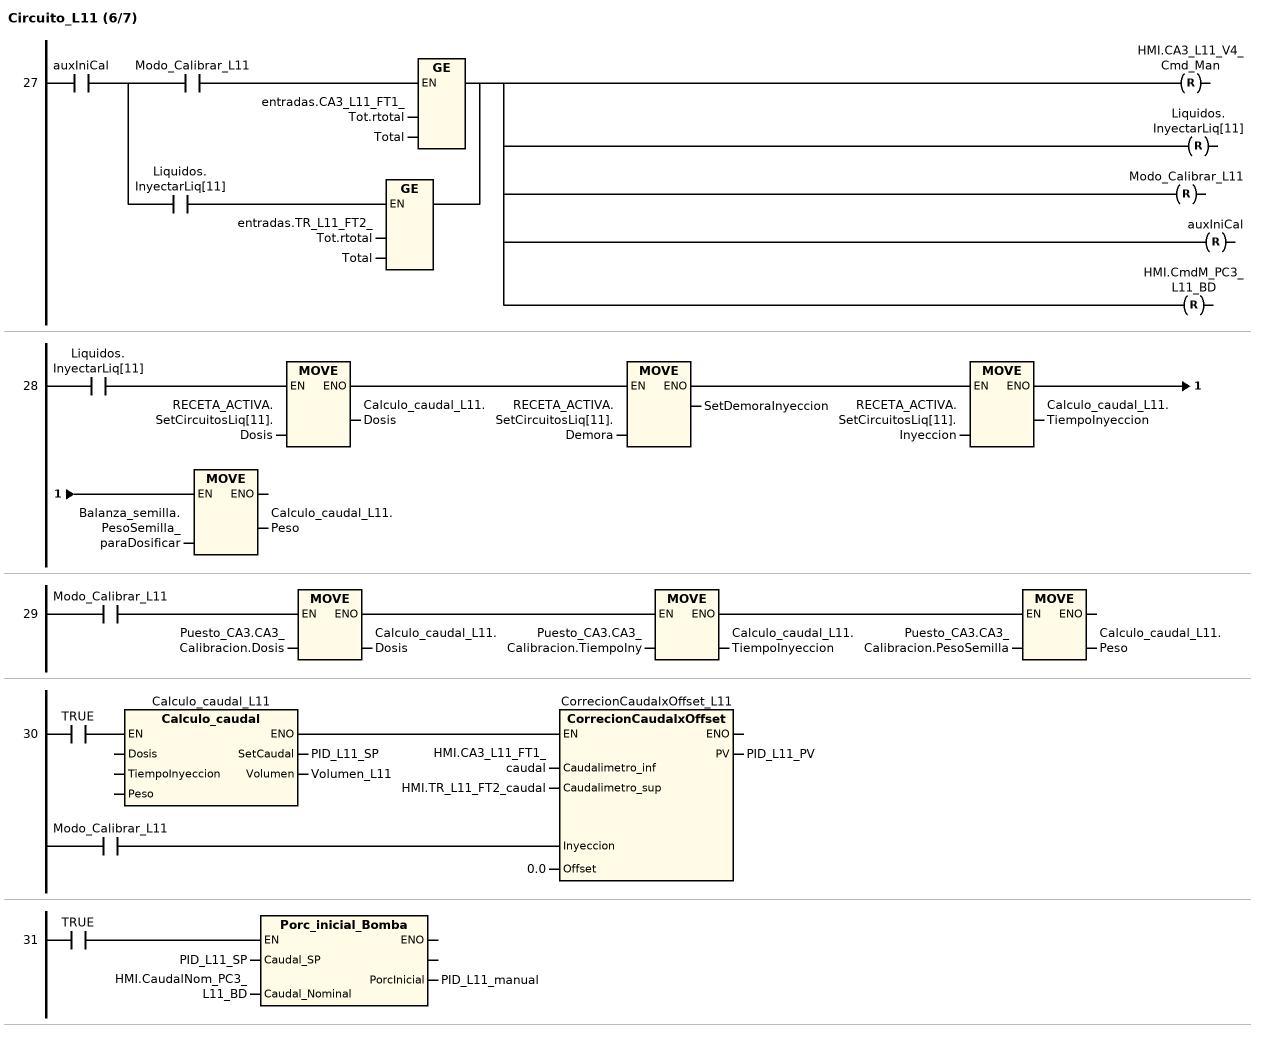
// NETWORK 27
_w10 := auxIniCal AND Modo_Calibrar_L11 AND entradas.CA3_L11_FT1_Tot.rtotal >= Total OR auxIniCal AND Liquidos.InyectarLiq[11] AND entradas.TR_L11_FT2_Tot.rtotal >= Total;
HMI.CA3_L11_V4_Cmd_Man R= _w10;
Liquidos.InyectarLiq[11] R= _w10;
Modo_Calibrar_L11 R= _w10;
auxIniCal R= _w10;
HMI.CmdM_PC3_L11_BD R= _w10;

// NETWORK 28
_w11 := Liquidos.InyectarLiq[11];
IF _w11 THEN Calculo_caudal_L11.Dosis := RECETA_ACTIVA.SetCircuitosLiq[11].Dosis; END_IF
IF _w11 THEN SetDemoraInyeccion := RECETA_ACTIVA.SetCircuitosLiq[11].Demora; END_IF
IF _w11 THEN Calculo_caudal_L11.TiempoInyeccion := RECETA_ACTIVA.SetCircuitosLiq[11].Inyeccion; END_IF
IF _w11 THEN Calculo_caudal_L11.Peso := Balanza_semilla.PesoSemilla_paraDosificar; END_IF

// NETWORK 29
_w12 := Modo_Calibrar_L11;
IF _w12 THEN Calculo_caudal_L11.Dosis := Puesto_CA3.CA3_Calibracion.Dosis; END_IF
IF _w12 THEN Calculo_caudal_L11.TiempoInyeccion := Puesto_CA3.CA3_Calibracion.TiempoIny; END_IF
IF _w12 THEN Calculo_caudal_L11.Peso := Puesto_CA3.CA3_Calibracion.PesoSemilla; END_IF

// NETWORK 30
Calculo_caudal_L11(SetCaudal => PID_L11_SP, Volumen => Volumen_L11); // Calculo_caudal
CorrecionCaudalxOffset_L11(
    Caudalimetro_inf := HMI.CA3_L11_FT1_caudal,
    Caudalimetro_sup := HMI.TR_L11_FT2_caudal,
    Inyeccion := Modo_Calibrar_L11,
    Offset := 0.0,
    PV => PID_L11_PV); // CorrecionCaudalxOffset

// NETWORK 31
Porc_inicial_Bomba(Caudal_SP := PID_L11_SP, Caudal_Nominal := HMI.CaudalNom_PC3_L11_BD, PorcInicial => PID_L11_manual);

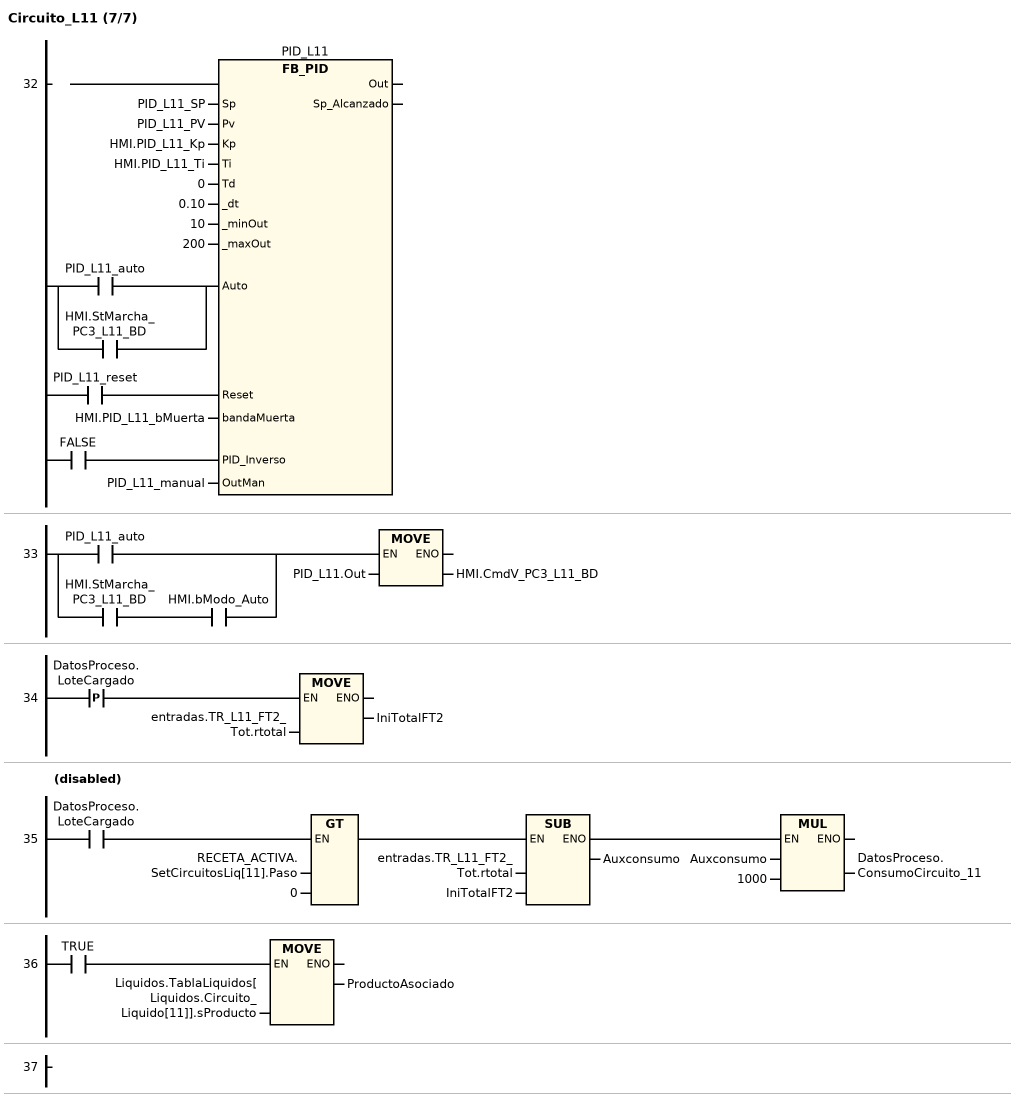
// NETWORK 32
PID_L11(
    Sp := PID_L11_SP,
    Pv := PID_L11_PV,
    Kp := HMI.PID_L11_Kp,
    Ti := HMI.PID_L11_Ti,
    Td := 0,
    _dt := 0.10,
    _minOut := 10,
    _maxOut := 200,
    Auto := PID_L11_auto OR HMI.StMarcha_PC3_L11_BD,
    Reset := PID_L11_reset,
    bandaMuerta := HMI.PID_L11_bMuerta,
    PID_Inverso := FALSE,
    OutMan := PID_L11_manual); // FB_PID

// NETWORK 33
IF PID_L11_auto OR HMI.StMarcha_PC3_L11_BD AND HMI.bModo_Auto THEN HMI.CmdV_PC3_L11_BD := PID_L11.Out; END_IF

// NETWORK 34
_rt2(CLK := DatosProceso.LoteCargado);
IF _rt2.Q THEN IniTotalFT2 := entradas.TR_L11_FT2_Tot.rtotal; END_IF

// NETWORK 35 (disabled)
// _w13 := DatosProceso.LoteCargado AND RECETA_ACTIVA.SetCircuitosLiq[11].Paso > 0;
// IF _w13 THEN Auxconsumo := entradas.TR_L11_FT2_Tot.rtotal - IniTotalFT2; END_IF
// IF _w13 THEN DatosProceso.ConsumoCircuito_11 := Auxconsumo * 1000; END_IF

// NETWORK 36
ProductoAsociado := Liquidos.TablaLiquidos[Liquidos.Circuito_Liquido[11]].sProducto;

// NETWORK 37

END_PROGRAM

// ---- POUs/Puesto_Calibracion_3/Circuito_L12.TcPOU
PROGRAM Circuito_L12
VAR_INPUT
	Modo_Calibrar_L12: BOOL;
END_VAR
VAR
	fbBomba_L12 :Equipo_Motor_ATV320;
	ControlValv_ioLink_V1:ControlValv_ioLink;
	ControlValv_ioLink_V2: ControlValv_ioLink;
	ControlValv_ioLink_V3: ControlValv_ioLink;
	ControlValv_ioLink_V4: ControlValv_ioLink;
	Falla_L12_V1:BOOL;
	Falla_L12_V2:BOOL;
	Falla_L12_V3:BOOL;
	Falla_L12_V4:BOOL;
	Balanza_PU3_WT12: Balanza;
	dHS:DINT;
	TOF_calibradoIBC: TOF;
	PID_L12_SP:REAL;
	PID_L12_auto:BOOL;
	PID_L12_reset:BOOL;
	PID_L12_manual:REAL;
	PID_L12_bMuerta:REAL := 5;
	PID_L12_Kp:REAL := 0.1;
	PID_L12_Ti:REAL := 100;
	PID_L12_PV:REAL;
	Dosis_L12:REAL;
	TiempoInyeccion_L12	:DINT;
	Peso	:REAL;
	Offset_L12:REAL;
	Inyeccion_L12:BOOL;

	Volumen_L12:REAL;
	Calculo_caudal_L12: Calculo_caudal;
	CorrecionCaudalxOffset_L12: CorrecionCaudalxOffset;
	tInyeccion: TON;
	Total :REAL;
	Totalant	:REAL;
	auxIniCal:BOOL;
	AuxVol12:REAL;
	TDemoraInyectar: TON;
	SetDemoraInyeccion: REAL;
	Tiempo_seg_to_TIME_DemoraInyec: Tiempo_seg_to_TIME;
	AuxTDemoraInyec: TIME;
	PID_L12: FB_PID;
	Tiempo_TIME_to_seg_InyCal: Tiempo_TIME_to_seg;
	AuxInyCal:TIME;
	IniTotalFT2:REAL;
	Auxconsumo:REAL;
	ProductoAsociado: STRING;
	Lavagem_Circuito12: Lavagem;
END_VAR

VAR PERSISTENT
	UltimaCalibracao	:UDINT;	//Data e hora da ultima calibração
END_VAR
VAR // added by the converter: edge detectors and wires of the graphical bodies
    _w1, _w2, _w3, _w4, _w5, _w6, _w7, _w8, _w9, _w10, _w11, _w12, _w13 : BOOL;
    _ft1 : F_TRIG;
    _rt1, _rt2 : R_TRIG;
END_VAR

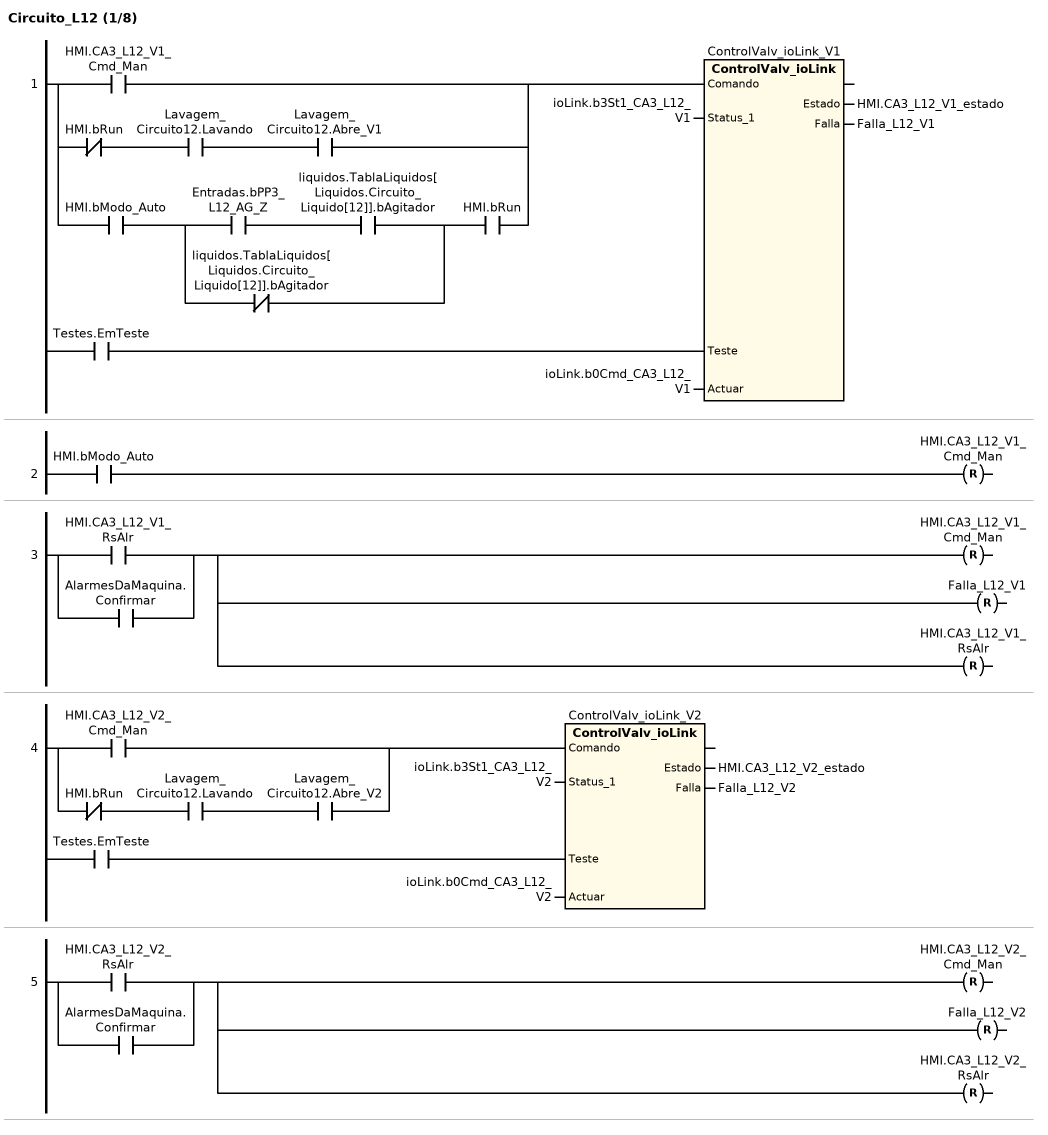
// NETWORK 1
ControlValv_ioLink_V1(
    Comando := HMI.CA3_L12_V1_Cmd_Man OR NOT HMI.bRun AND Lavagem_Circuito12.Lavando AND Lavagem_Circuito12.Abre_V1 OR HMI.bModo_Auto AND (Entradas.bPP3_L12_AG_Z AND (liquidos.TablaLiquidos[Liquidos.Circuito_Liquido[12]].bAgitador) OR NOT (liquidos.TablaLiquidos[Liquidos.Circuito_Liquido[12]].bAgitador)) AND HMI.bRun,
    Status_1 := ioLink.b3St1_CA3_L12_V1,
    Teste := Testes.EmTeste,
    Actuar := ioLink.b0Cmd_CA3_L12_V1,
    Estado => HMI.CA3_L12_V1_estado,
    Falla => Falla_L12_V1); // ControlValv_ioLink

// NETWORK 2
HMI.CA3_L12_V1_Cmd_Man R= HMI.bModo_Auto;

// NETWORK 3
_w1 := HMI.CA3_L12_V1_RsAlr OR AlarmesDaMaquina.Confirmar;
HMI.CA3_L12_V1_Cmd_Man R= _w1;
Falla_L12_V1 R= _w1;
HMI.CA3_L12_V1_RsAlr R= _w1;

// NETWORK 4
ControlValv_ioLink_V2(
    Comando := HMI.CA3_L12_V2_Cmd_Man OR NOT HMI.bRun AND Lavagem_Circuito12.Lavando AND Lavagem_Circuito12.Abre_V2,
    Status_1 := ioLink.b3St1_CA3_L12_V2,
    Teste := Testes.EmTeste,
    Actuar := ioLink.b0Cmd_CA3_L12_V2,
    Estado => HMI.CA3_L12_V2_estado,
    Falla => Falla_L12_V2); // ControlValv_ioLink

// NETWORK 5
_w2 := HMI.CA3_L12_V2_RsAlr OR AlarmesDaMaquina.Confirmar;
HMI.CA3_L12_V2_Cmd_Man R= _w2;
Falla_L12_V2 R= _w2;
HMI.CA3_L12_V2_RsAlr R= _w2;

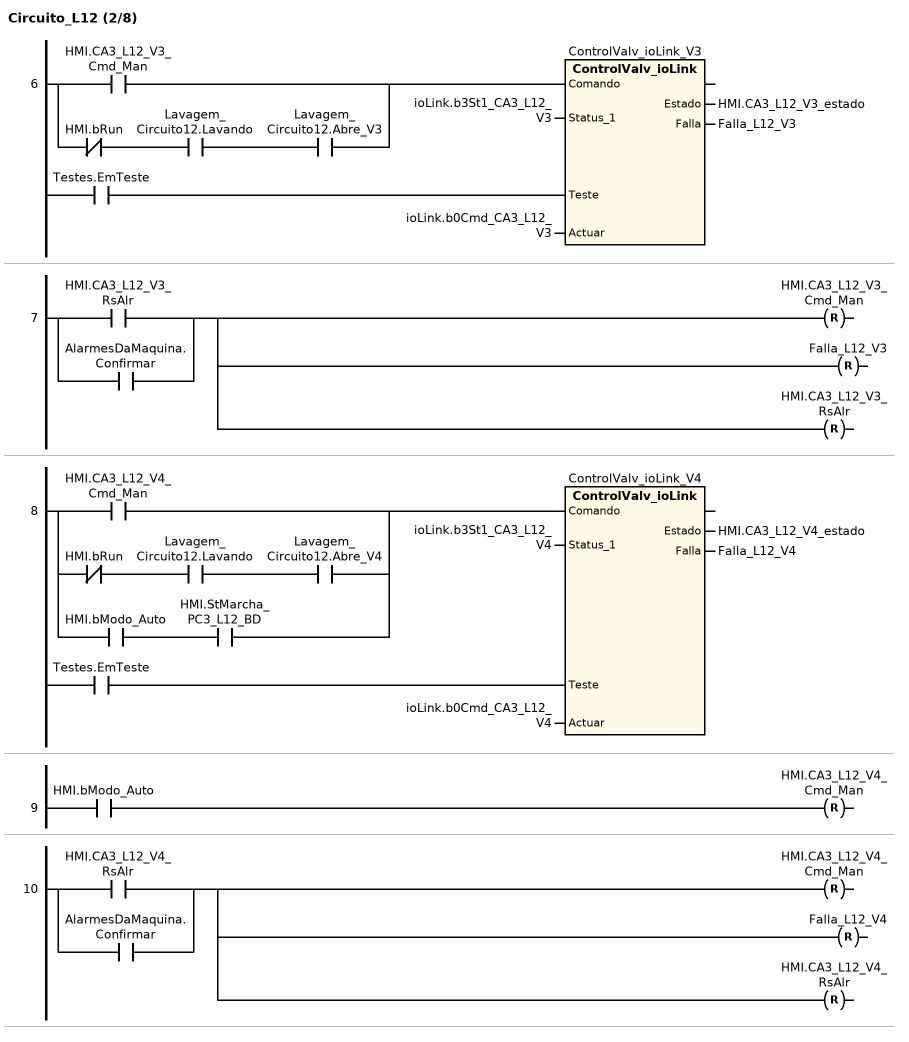
// NETWORK 6
ControlValv_ioLink_V3(
    Comando := HMI.CA3_L12_V3_Cmd_Man OR NOT HMI.bRun AND Lavagem_Circuito12.Lavando AND Lavagem_Circuito12.Abre_V3,
    Status_1 := ioLink.b3St1_CA3_L12_V3,
    Teste := Testes.EmTeste,
    Actuar := ioLink.b0Cmd_CA3_L12_V3,
    Estado => HMI.CA3_L12_V3_estado,
    Falla => Falla_L12_V3); // ControlValv_ioLink

// NETWORK 7
_w3 := HMI.CA3_L12_V3_RsAlr OR AlarmesDaMaquina.Confirmar;
HMI.CA3_L12_V3_Cmd_Man R= _w3;
Falla_L12_V3 R= _w3;
HMI.CA3_L12_V3_RsAlr R= _w3;

// NETWORK 8
ControlValv_ioLink_V4(
    Comando := HMI.CA3_L12_V4_Cmd_Man OR NOT HMI.bRun AND Lavagem_Circuito12.Lavando AND Lavagem_Circuito12.Abre_V4 OR HMI.bModo_Auto AND HMI.StMarcha_PC3_L12_BD,
    Status_1 := ioLink.b3St1_CA3_L12_V4,
    Teste := Testes.EmTeste,
    Actuar := ioLink.b0Cmd_CA3_L12_V4,
    Estado => HMI.CA3_L12_V4_estado,
    Falla => Falla_L12_V4); // ControlValv_ioLink

// NETWORK 9
HMI.CA3_L12_V4_Cmd_Man R= HMI.bModo_Auto;

// NETWORK 10
_w4 := HMI.CA3_L12_V4_RsAlr OR AlarmesDaMaquina.Confirmar;
HMI.CA3_L12_V4_Cmd_Man R= _w4;
Falla_L12_V4 R= _w4;
HMI.CA3_L12_V4_RsAlr R= _w4;

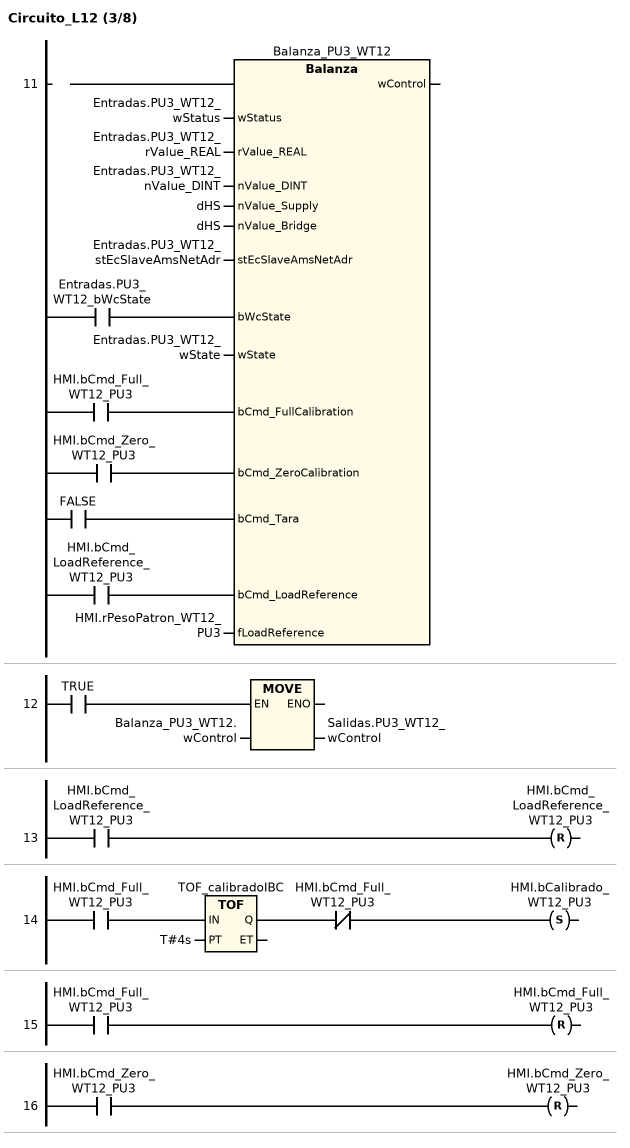
// NETWORK 11
Balanza_PU3_WT12(
    wStatus := Entradas.PU3_WT12_wStatus,
    rValue_REAL := Entradas.PU3_WT12_rValue_REAL,
    nValue_DINT := Entradas.PU3_WT12_nValue_DINT,
    nValue_Supply := dHS,
    nValue_Bridge := dHS,
    stEcSlaveAmsNetAdr := Entradas.PU3_WT12_stEcSlaveAmsNetAdr,
    bWcState := Entradas.PU3_WT12_bWcState,
    wState := Entradas.PU3_WT12_wState,
    bCmd_FullCalibration := HMI.bCmd_Full_WT12_PU3,
    bCmd_ZeroCalibration := HMI.bCmd_Zero_WT12_PU3,
    bCmd_Tara := FALSE,
    bCmd_LoadReference := HMI.bCmd_LoadReference_WT12_PU3,
    fLoadReference := HMI.rPesoPatron_WT12_PU3); // Balanza

// NETWORK 12
Salidas.PU3_WT12_wControl := Balanza_PU3_WT12.wControl;

// NETWORK 13
HMI.bCmd_LoadReference_WT12_PU3 R= HMI.bCmd_LoadReference_WT12_PU3;

// NETWORK 14
TOF_calibradoIBC(IN := HMI.bCmd_Full_WT12_PU3, PT := T#4s); // TOF
HMI.bCalibrado_WT12_PU3 S= TOF_calibradoIBC.Q AND NOT HMI.bCmd_Full_WT12_PU3;

// NETWORK 15
HMI.bCmd_Full_WT12_PU3 R= HMI.bCmd_Full_WT12_PU3;

// NETWORK 16
HMI.bCmd_Zero_WT12_PU3 R= HMI.bCmd_Zero_WT12_PU3;

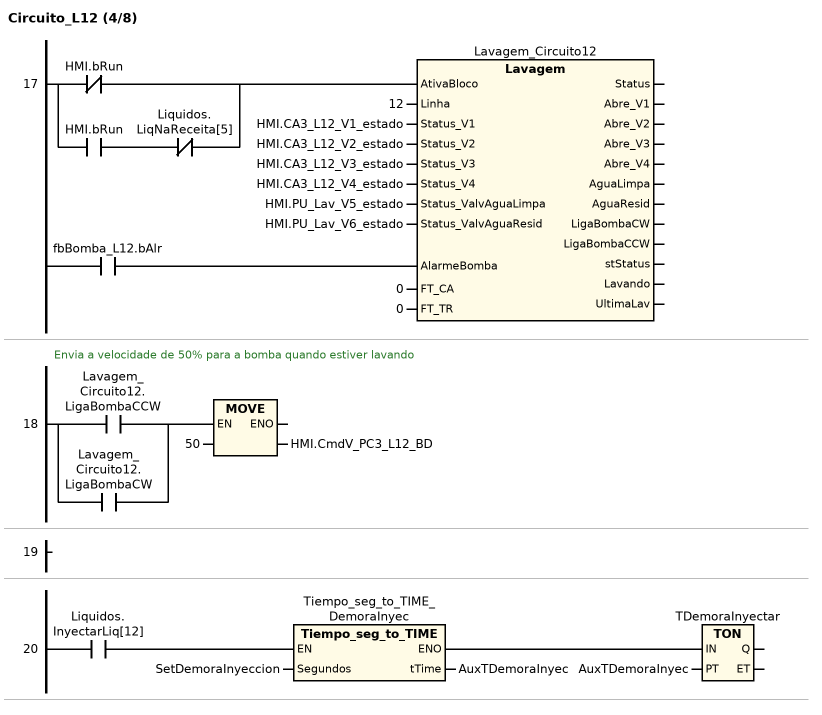
// NETWORK 17
Lavagem_Circuito12(
    AtivaBloco := NOT HMI.bRun OR HMI.bRun AND NOT Liquidos.LiqNaReceita[5],
    Linha := 12,
    Status_V1 := HMI.CA3_L12_V1_estado,
    Status_V2 := HMI.CA3_L12_V2_estado,
    Status_V3 := HMI.CA3_L12_V3_estado,
    Status_V4 := HMI.CA3_L12_V4_estado,
    Status_ValvAguaLimpa := HMI.PU_Lav_V5_estado,
    Status_ValvAguaResid := HMI.PU_Lav_V6_estado,
    AlarmeBomba := fbBomba_L12.bAlr,
    FT_CA := 0,
    FT_TR := 0); // Lavagem

// NETWORK 18
// Envia a velocidade de 50% para a bomba quando estiver lavando
IF Lavagem_Circuito12.LigaBombaCCW OR Lavagem_Circuito12.LigaBombaCW THEN HMI.CmdV_PC3_L12_BD := 50; END_IF

// NETWORK 19

// NETWORK 20
_w5 := Liquidos.InyectarLiq[12];
IF _w5 THEN
    Tiempo_seg_to_TIME_DemoraInyec(Segundos := SetDemoraInyeccion, tTime => AuxTDemoraInyec); // Tiempo_seg_to_TIME
END_IF
TDemoraInyectar(IN := _w5, PT := AuxTDemoraInyec); // TON

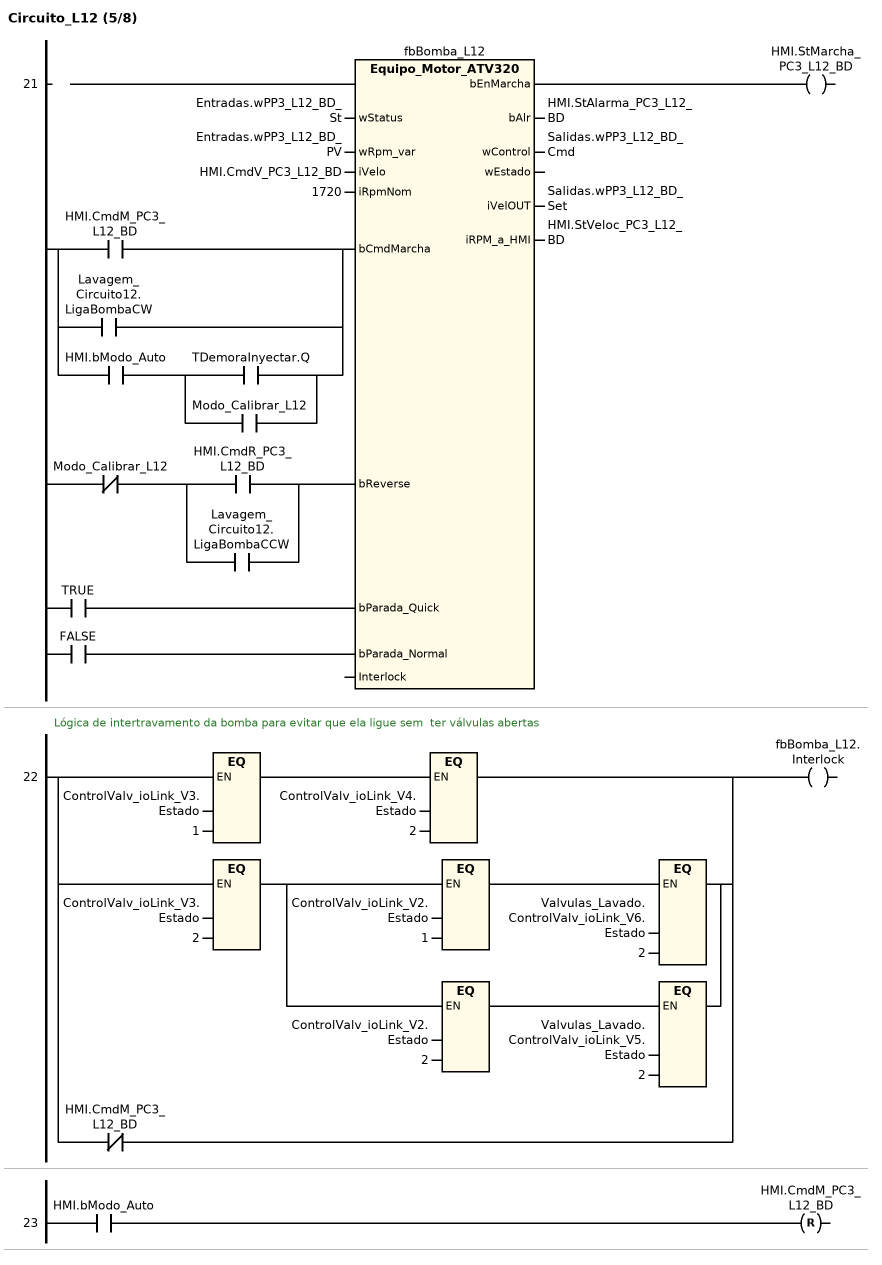
// NETWORK 21
fbBomba_L12(
    wStatus := Entradas.wPP3_L12_BD_St,
    wRpm_var := Entradas.wPP3_L12_BD_PV,
    iVelo := HMI.CmdV_PC3_L12_BD,
    iRpmNom := 1720,
    bCmdMarcha := HMI.CmdM_PC3_L12_BD OR Lavagem_Circuito12.LigaBombaCW OR HMI.bModo_Auto AND (TDemoraInyectar.Q OR Modo_Calibrar_L12),
    bReverse := NOT Modo_Calibrar_L12 AND (HMI.CmdR_PC3_L12_BD OR Lavagem_Circuito12.LigaBombaCCW),
    bParada_Quick := TRUE,
    bParada_Normal := FALSE,
    bAlr => HMI.StAlarma_PC3_L12_BD,
    wControl => Salidas.wPP3_L12_BD_Cmd,
    iVelOUT => Salidas.wPP3_L12_BD_Set,
    iRPM_a_HMI => HMI.StVeloc_PC3_L12_BD); // Equipo_Motor_ATV320
HMI.StMarcha_PC3_L12_BD := fbBomba_L12.bEnMarcha;

// NETWORK 22
// Lógica de intertravamento da bomba para evitar que ela ligue sem  ter válvulas abertas
_w6 := NOT HMI.CmdM_PC3_L12_BD;
IF NOT _w6 THEN
    _w7 := ControlValv_ioLink_V3.Estado = 2;
    _w6 := ControlValv_ioLink_V3.Estado = 1 AND ControlValv_ioLink_V4.Estado = 2 OR (_w7 AND ControlValv_ioLink_V2.Estado = 1 AND Valvulas_Lavado.ControlValv_ioLink_V6.Estado = 2 OR _w7 AND ControlValv_ioLink_V2.Estado = 2 AND Valvulas_Lavado.ControlValv_ioLink_V5.Estado = 2);
END_IF
fbBomba_L12.Interlock := _w6;

// NETWORK 23
HMI.CmdM_PC3_L12_BD R= HMI.bModo_Auto;

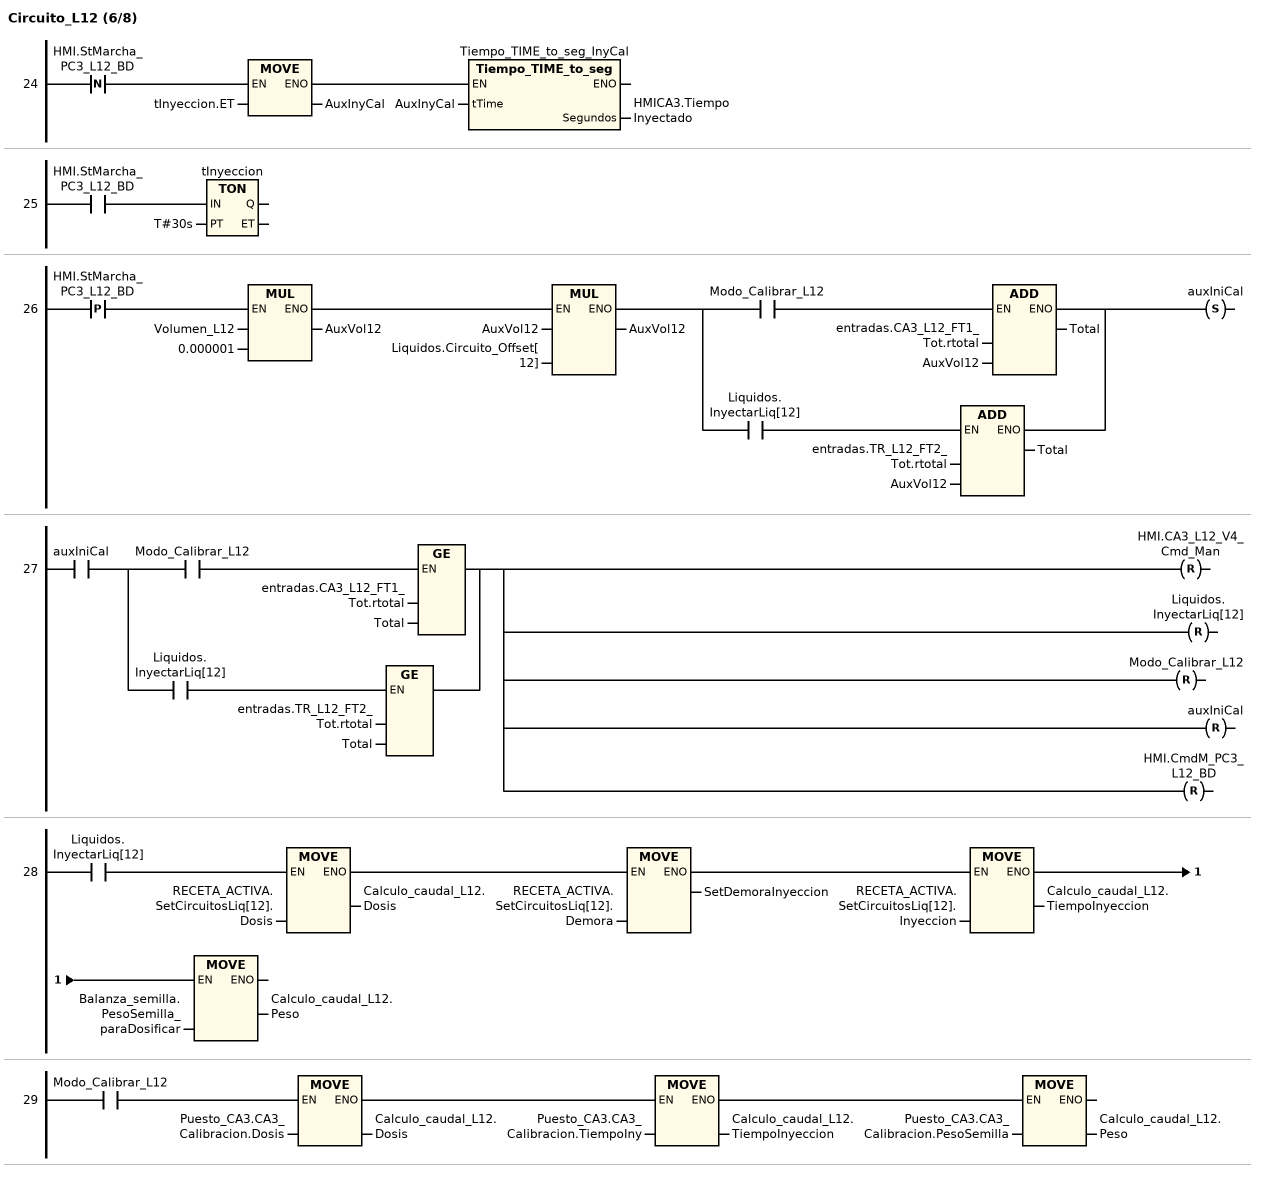
// NETWORK 24
_ft1(CLK := HMI.StMarcha_PC3_L12_BD);
_w8 := _ft1.Q;
IF _w8 THEN AuxInyCal := tInyeccion.ET; END_IF
IF _w8 THEN
    Tiempo_TIME_to_seg_InyCal(tTime := AuxInyCal, Segundos => HMICA3.TiempoInyectado); // Tiempo_TIME_to_seg
END_IF

// NETWORK 25
tInyeccion(IN := HMI.StMarcha_PC3_L12_BD, PT := T#30s); // TON

// NETWORK 26
_rt1(CLK := HMI.StMarcha_PC3_L12_BD);
_w9 := _rt1.Q;
IF _w9 THEN AuxVol12 := Volumen_L12 * 0.000001; END_IF
IF _w9 THEN AuxVol12 := AuxVol12 * Liquidos.Circuito_Offset[12]; END_IF
IF _w9 AND Modo_Calibrar_L12 THEN Total := entradas.CA3_L12_FT1_Tot.rtotal + AuxVol12; END_IF
IF _w9 AND Liquidos.InyectarLiq[12] THEN Total := entradas.TR_L12_FT2_Tot.rtotal + AuxVol12; END_IF
auxIniCal S= _w9 AND Modo_Calibrar_L12 OR _w9 AND Liquidos.InyectarLiq[12];

// NETWORK 27
_w10 := auxIniCal AND Modo_Calibrar_L12 AND entradas.CA3_L12_FT1_Tot.rtotal >= Total OR auxIniCal AND Liquidos.InyectarLiq[12] AND entradas.TR_L12_FT2_Tot.rtotal >= Total;
HMI.CA3_L12_V4_Cmd_Man R= _w10;
Liquidos.InyectarLiq[12] R= _w10;
Modo_Calibrar_L12 R= _w10;
auxIniCal R= _w10;
HMI.CmdM_PC3_L12_BD R= _w10;

// NETWORK 28
_w11 := Liquidos.InyectarLiq[12];
IF _w11 THEN Calculo_caudal_L12.Dosis := RECETA_ACTIVA.SetCircuitosLiq[12].Dosis; END_IF
IF _w11 THEN SetDemoraInyeccion := RECETA_ACTIVA.SetCircuitosLiq[12].Demora; END_IF
IF _w11 THEN Calculo_caudal_L12.TiempoInyeccion := RECETA_ACTIVA.SetCircuitosLiq[12].Inyeccion; END_IF
IF _w11 THEN Calculo_caudal_L12.Peso := Balanza_semilla.PesoSemilla_paraDosificar; END_IF

// NETWORK 29
_w12 := Modo_Calibrar_L12;
IF _w12 THEN Calculo_caudal_L12.Dosis := Puesto_CA3.CA3_Calibracion.Dosis; END_IF
IF _w12 THEN Calculo_caudal_L12.TiempoInyeccion := Puesto_CA3.CA3_Calibracion.TiempoIny; END_IF
IF _w12 THEN Calculo_caudal_L12.Peso := Puesto_CA3.CA3_Calibracion.PesoSemilla; END_IF

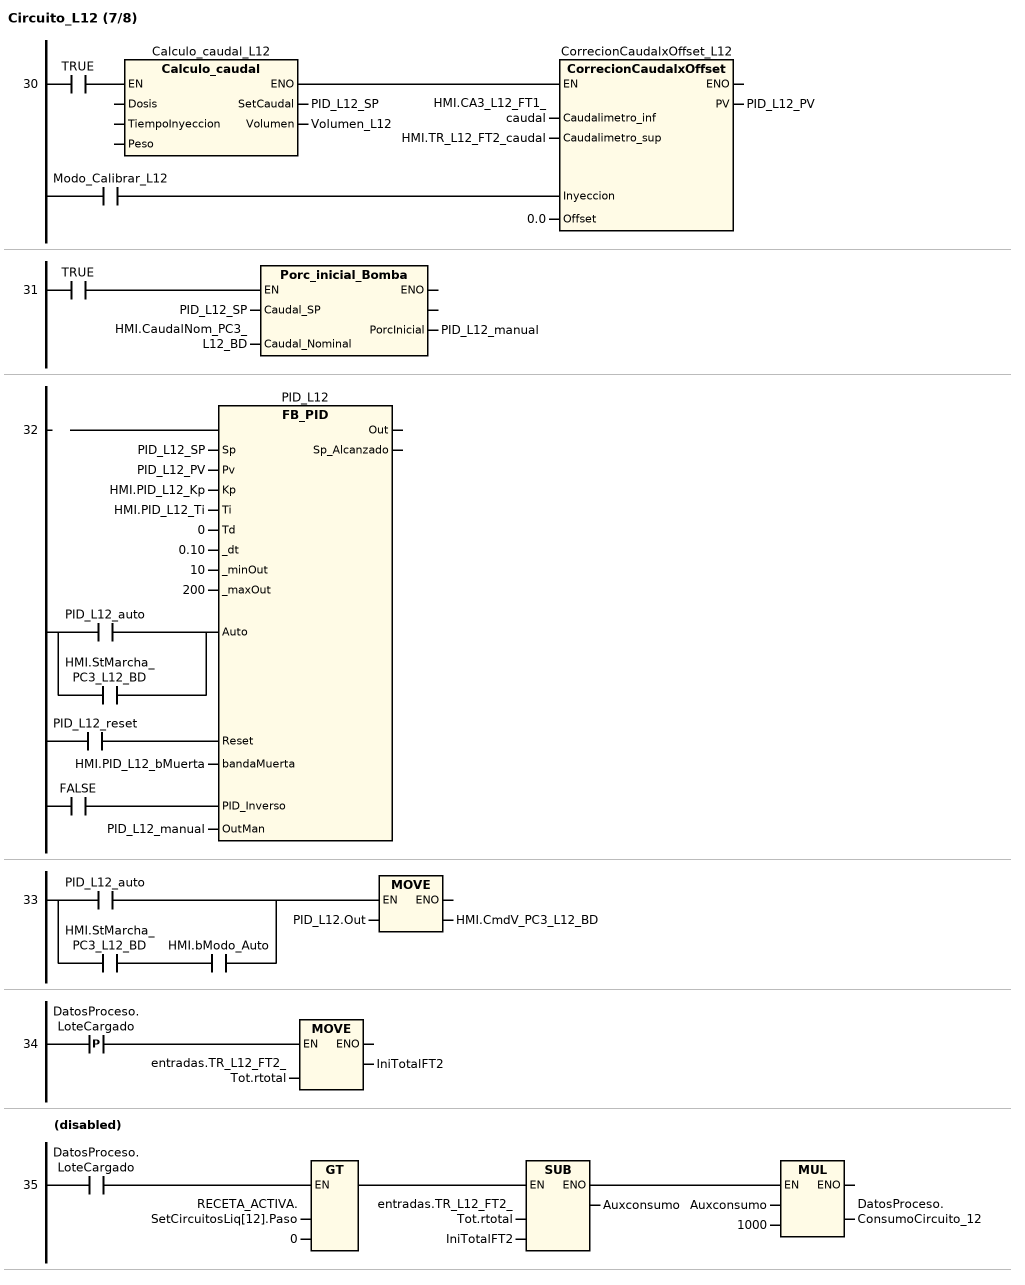
// NETWORK 30
Calculo_caudal_L12(SetCaudal => PID_L12_SP, Volumen => Volumen_L12); // Calculo_caudal
CorrecionCaudalxOffset_L12(
    Caudalimetro_inf := HMI.CA3_L12_FT1_caudal,
    Caudalimetro_sup := HMI.TR_L12_FT2_caudal,
    Inyeccion := Modo_Calibrar_L12,
    Offset := 0.0,
    PV => PID_L12_PV); // CorrecionCaudalxOffset

// NETWORK 31
Porc_inicial_Bomba(Caudal_SP := PID_L12_SP, Caudal_Nominal := HMI.CaudalNom_PC3_L12_BD, PorcInicial => PID_L12_manual);

// NETWORK 32
PID_L12(
    Sp := PID_L12_SP,
    Pv := PID_L12_PV,
    Kp := HMI.PID_L12_Kp,
    Ti := HMI.PID_L12_Ti,
    Td := 0,
    _dt := 0.10,
    _minOut := 10,
    _maxOut := 200,
    Auto := PID_L12_auto OR HMI.StMarcha_PC3_L12_BD,
    Reset := PID_L12_reset,
    bandaMuerta := HMI.PID_L12_bMuerta,
    PID_Inverso := FALSE,
    OutMan := PID_L12_manual); // FB_PID

// NETWORK 33
IF PID_L12_auto OR HMI.StMarcha_PC3_L12_BD AND HMI.bModo_Auto THEN HMI.CmdV_PC3_L12_BD := PID_L12.Out; END_IF

// NETWORK 34
_rt2(CLK := DatosProceso.LoteCargado);
IF _rt2.Q THEN IniTotalFT2 := entradas.TR_L12_FT2_Tot.rtotal; END_IF

// NETWORK 35 (disabled)
// _w13 := DatosProceso.LoteCargado AND RECETA_ACTIVA.SetCircuitosLiq[12].Paso > 0;
// IF _w13 THEN Auxconsumo := entradas.TR_L12_FT2_Tot.rtotal - IniTotalFT2; END_IF
// IF _w13 THEN DatosProceso.ConsumoCircuito_12 := Auxconsumo * 1000; END_IF

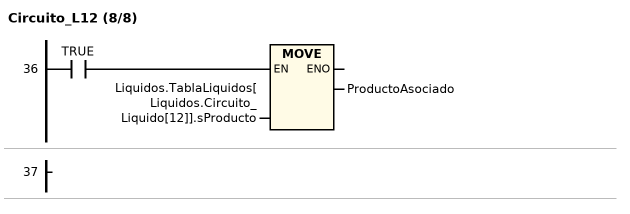
// NETWORK 36
ProductoAsociado := Liquidos.TablaLiquidos[Liquidos.Circuito_Liquido[12]].sProducto;

// NETWORK 37

END_PROGRAM

// ---- POUs/Perifericos/Carga_semilla.TcPOU
PROGRAM Carga_semilla
VAR
	
	fbPE_H_VF1 :Equipo_Motor_ATV320;	//Elevador TRBB	
	fbPE_H_VF2 :Equipo_Motor_ATV320;	//Elevador carga tratadora
	Demora_PE_H_HLS: TON;
	Demora_TR_S_HLS: TON;
	ParadaPE_H_VF1: TOF;
	ParadaPE_TR_S_HLS: TOF;
	TmrDemoraPE_H_VF2: TOF;
	TmrDemoraPE_H_VF1: TOF;
	Tiempo_seg_to_TIME_PE_H_VF1: Tiempo_seg_to_TIME;
	Tiempo_seg_to_TIME_PE_H_VF2: Tiempo_seg_to_TIME;
	TDemoraTR_S_V7: TON;
	TDemoraTR_S_V8: TON;
END_VAR
VAR // added by the converter: edge detectors and wires of the graphical bodies
    _w1, _w2, _w3 : BOOL;
    _ft1, _ft2 : F_TRIG;
END_VAR

